// TwinCAT 3 PLC project Controller
// Title: BIO2
// Company: 3P Innovation Ltd.
// Author: James Tyler
// ProgramVersion: 3.1.0.8
// libraries:
//   Standard, * (System)
//   Tc2_ControllerToolbox, * (Beckhoff Automation GmbH)
//   Tc2_Standard, * (Beckhoff Automation GmbH)
//   Tc2_System, * (Beckhoff Automation GmbH)
//   Tc2_TempController, * (Beckhoff Automation GmbH)
//   Tc2_Utilities, * (Beckhoff Automation GmbH)
//   Tc2_XmlDataSrv, * (Beckhoff Automation GmbH)
//   Tc3_Interfaces, * (Beckhoff Automation GmbH)
//   Tc3_Module, * (Beckhoff Automation GmbH)
//   Tc_Persistent, * (Red Rock Controls Limited)
//   Tc2_MC2,newest,Beckhoff Automation GmbH
//   Tc_Collections,1.0.0.8,Red Rock Controls
//   Tc_Helper,1.0.0.8,Red Rock Controls
// project tree:
//   Classes/Compress/ FB_Compress.TcPOU
//   Classes/Config/ TConfig.TcPOU, TConfigData.TcDUT
//   Classes/Pusher/ FB_Pusher.TcPOU
//   Classes/Shield/ FB_Shield.TcPOU
//   DUTs/ E_LampState.TcDUT (not stored), E_CTRL_STATE.TcDUT, Limits.TcDUT, Recipe.TcDUT, Rec_Compress.TcDUT, Rec_Other.TcDUT, Rec_Pusher.TcDUT, Rec_Clamp.TcDUT (not stored), Rec_Shield.TcDUT
//   GVLs/ GVL_IO.TcGVL, GVL_Objects.TcGVL, GVL_ZenOn.TcGVL
//   / PlcTask.TcTTO, Task_Fast.TcTTO
//   POUs/ Config_Slow.TcPOU, FB_AxisControl.TcPOU, FB_LampController.TcPOU, F_DisplayText.TcPOU (not stored), PRG_MAIN.TcPOU, PRG_IO.TcPOU, PRG_Machine.TcPOU
//   XML/ eXMLState.TcDUT, FB_Retain.TcPOU, FB_RetainedData.TcPOU (not stored)
// real-time tasks:
//   TASK PlcTask: cycle T#10ms, priority 20, ADS port 350
//   TASK Task_Fast: cycle T#1ms, priority 21, ADS port 351
// motion (NC):
//   TASK NC-Task 1 SAF: cycle T#2ms, priority 4, ADS port 501
//   TASK NC-Task 1 SVB: cycle T#10ms, priority 8, ADS port 511
//   AXIS Compress (id 1)
//     Dynamic: Acceleration=60.7875, Deceleration=60.7875, Jerk=182.363
//     Velo: RefSearch=0.40525, RefSync=0.40525, SlowManual=2.02625, FastManual=12.1575, Fast=40.525, Maximum=200
//     OtherSettings: AllowMotionCmdToSlave=true
//     encoder EncType=19
//       EncPara: ScaleFactorNumerator=0.5, ScaleFactorDenominator=1048576, ModuloFactor=0.5, MaxCount=#xffffffff
//     drive DrvType=16
//       DrvPara: MaxCount=#xffffffff
//         Analog: VeloReferenz=200, VeloScale=32
//         TimeComp: TaskDelayCycles=1
//     controller CtrType=1
//       CtrPara: PriorControlFactor=1
//         PosDiffControl: Enable=false, Range=0.05
//         PID: PosKp=20
//         Observer: BandWidth=20
//   AXIS Pusher (id 2)
//     Dynamic: Acceleration=60.7875, Deceleration=60.7875, Jerk=182.3625
//     Velo: RefSearch=0.40525, RefSync=0.40525, SlowManual=2.02625, FastManual=12.1575, Fast=40.525, Maximum=40.525
//     OtherSettings: AllowMotionCmdToSlave=true
//     encoder EncType=19
//       EncPara: ScaleFactorNumerator=0.5, ScaleFactorDenominator=1048576, ModuloFactor=0.5, MaxCount=#xffffffff
//     drive DrvType=16
//       DrvPara: MaxCount=#xffffffff
//         Analog: VeloReferenz=100, VeloScale=32
//         TimeComp: TaskDelayCycles=1
//     controller CtrType=1
//       CtrPara: PriorControlFactor=1
//         PosDiffControl: Enable=false, Range=0.5
//         PID: PosKp=20
//         Observer: BandWidth=20
//   AXIS Shield (id 3)
//     Dynamic: Acceleration=60.7875, Deceleration=60.7875, Jerk=182.363
//     Velo: RefSearch=0.40525, RefSync=0.40525, SlowManual=2.02625, FastManual=12.1575, Fast=200, Maximum=200
//     OtherSettings: AllowMotionCmdToSlave=true
//     encoder EncType=19
//       EncPara: ScaleFactorNumerator=0.5, ScaleFactorDenominator=1048576, ModuloFactor=0.5, MaxCount=#xffffffff
//     drive DrvType=16
//       DrvPara: MaxCount=#xffffffff
//         Analog: VeloReferenz=200, VeloScale=32
//         TimeComp: TaskDelayCycles=1
//     controller CtrType=1
//       CtrPara: PriorControlFactor=1
//         PosDiffControl: Enable=false, Range=0.05
//         PID: PosKp=20
//         Observer: BandWidth=20
// I/O:
//   DEVICE Device 1 (EtherCAT), AmsNetId 5.47.207.20.2.1
//     Term 5 (EK1100) [EK1100 EtherCAT Coupler (2A E-Bus)]
//       Term 6 (EL1809) [EL1809 16Ch. Dig. Input 24V, 3ms]
//       Term 7 (EL2798) [EL2798 8Ch. Dig. Output 24V AC/DC, 2A, potential-free]
//       Term 13 (EL9011) [EL9011 End Terminal]
//     Term 8 (EK1100) [EK1100 EtherCAT Coupler (2A E-Bus)]
//       Term 9 (EL7201-9014) [EL7201-9014 1Ch. MDP742 Servo motor output stage with OCT (50V, 4A) and STO input]
//       Term 10 (EL7201-9014) [EL7201-9014 1Ch. MDP742 Servo motor output stage with OCT (50V, 4A)  and STO input]
//       Term 11 (EL7201-9014) [EL7201-9014 1Ch. MDP742 Servo motor output stage with OCT (50V, 4A)  and STO input]
//       Term 12 (EL1809) [EL1809 16Ch. Dig. Input 24V, 3ms]
//       Term 14 (EL9011) [EL9011 End Terminal]
//   DEVICE Device 3 (RT-Ethernet Protocol) (disabled), AmsNetId 5.47.207.20.4.1
// variable links:
//   NC-Task 1 SAF/Axes/Compress <-> Device 1 (EtherCAT)/Term 8 (EK1100)/Term 9 (EL7201-9014)
//     Drive/Inputs/In/nDcOutputTime <-> InfoData/DcOutputShift
//     Drive/Inputs/In/nState1 <-> DRV Statusword/Statusword
//     Drive/Inputs/In/nState2 <-> DRV Statusword/Statusword @bit 8
//     Drive/Inputs/In/nState4 @bit 1 <-> WcState/InputToggle
//     Drive/Inputs/In/nState4 <-> WcState/WcState
//     Drive/Outputs/Out/nCtrl1 <-> DRV Controlword/Controlword
//     Drive/Outputs/Out/nCtrl2 <-> DRV Controlword/Controlword @bit 8
//     Drive/Outputs/Out/nDataOut2 <-> DRV Target velocity/Target velocity
//     Enc/Inputs/In/nDataIn1 <-> FB Position/Position
//     Enc/Inputs/In/nDcInputTime <-> InfoData/DcInputShift
//     Enc/Inputs/In/nState4 @bit 1 <-> WcState/InputToggle
//     Enc/Inputs/In/nState4 <-> WcState/WcState
//   NC-Task 1 SAF/Axes/Pusher <-> Device 1 (EtherCAT)/Term 8 (EK1100)/Term 10 (EL7201-9014)
//     Drive/Inputs/In/nDcOutputTime <-> InfoData/DcOutputShift
//     Drive/Inputs/In/nState1 <-> DRV Statusword/Statusword
//     Drive/Inputs/In/nState2 <-> DRV Statusword/Statusword @bit 8
//     Drive/Inputs/In/nState4 @bit 1 <-> WcState/InputToggle
//     Drive/Inputs/In/nState4 <-> WcState/WcState
//     Drive/Outputs/Out/nCtrl1 <-> DRV Controlword/Controlword
//     Drive/Outputs/Out/nCtrl2 <-> DRV Controlword/Controlword @bit 8
//     Drive/Outputs/Out/nDataOut2 <-> DRV Target velocity/Target velocity
//     Enc/Inputs/In/nDataIn1 <-> FB Position/Position
//     Enc/Inputs/In/nDcInputTime <-> InfoData/DcInputShift
//     Enc/Inputs/In/nState4 @bit 1 <-> WcState/InputToggle
//     Enc/Inputs/In/nState4 <-> WcState/WcState
//   NC-Task 1 SAF/Axes/Shield <-> Device 1 (EtherCAT)/Term 8 (EK1100)/Term 11 (EL7201-9014)
//     Drive/Inputs/In/nDcOutputTime <-> InfoData/DcOutputShift
//     Drive/Inputs/In/nState1 <-> DRV Statusword/Statusword
//     Drive/Inputs/In/nState2 <-> DRV Statusword/Statusword @bit 8
//     Drive/Inputs/In/nState4 @bit 1 <-> WcState/InputToggle
//     Drive/Inputs/In/nState4 <-> WcState/WcState
//     Drive/Outputs/Out/nCtrl1 <-> DRV Controlword/Controlword
//     Drive/Outputs/Out/nCtrl2 <-> DRV Controlword/Controlword @bit 8
//     Drive/Outputs/Out/nDataOut2 <-> DRV Target velocity/Target velocity
//     Enc/Inputs/In/nDataIn1 <-> FB Position/Position
//     Enc/Inputs/In/nDcInputTime <-> InfoData/DcInputShift
//     Enc/Inputs/In/nState4 @bit 1 <-> WcState/InputToggle
//     Enc/Inputs/In/nState4 <-> WcState/WcState
//   Controller/Controller Instance <-> Device 1 (EtherCAT)/Term 5 (EK1100)/Term 6 (EL1809)
//     PlcTask Inputs/GVL_IO.ixCabinetE_StopButtonOkay <-> Channel 1/Cabinet E-Stop
//     PlcTask Inputs/GVL_IO.ixE_StopRelayOkay <-> Channel 2/Input
//     PlcTask Inputs/GVL_IO.ixGuardRelayOkay <-> Channel 3/Input
//     PlcTask Inputs/GVL_IO.ixResetButton <-> Channel 6/Input
//     PlcTask Inputs/GVL_IO.ixStartButton <-> Channel 9/Input
//     PlcTask Inputs/GVL_IO.ixStop_Button <-> Channel 10/Input
//     Task_Fast Inputs/GVL_IO.ixSpareIN4 <-> Channel 4/Input
//     Task_Fast Inputs/GVL_IO.ixSpareIN5 <-> Channel 5/Input
//     Task_Fast Inputs/GVL_IO.ixSpareIN7 <-> Channel 7/Input
//     Task_Fast Inputs/GVL_IO.ixSpareIN8 <-> Channel 8/Input
//   Controller/Controller Instance <-> Device 1 (EtherCAT)/Term 5 (EK1100)/Term 7 (EL2798)
//     PlcTask Outputs/GVL_IO.qxClamp <-> Channel 2/Output
//     PlcTask Outputs/GVL_IO.qxEnableE_Stop <-> Channel 1/Output
//     PlcTask Outputs/GVL_IO.qxResetButtonLamp <-> Channel 5/Output
//     PlcTask Outputs/GVL_IO.qxStartButtonLamp <-> Channel 4/Output
//     Task_Fast Outputs/GVL_IO.qxSpareOUT3 <-> Channel 3/Output
//   Controller/Controller Instance <-> Device 1 (EtherCAT)/Term 8 (EK1100)/Term 12 (EL1809)
//     PlcTask Inputs/GVL_IO.ixCompressHomeSwitch <-> Channel 1/Input
//     PlcTask Inputs/GVL_IO.ixGuardOkay <-> Channel 9/Input
//     PlcTask Inputs/GVL_IO.ixMachineE_StopButtonOkay <-> Channel 10/Input
//     PlcTask Inputs/GVL_IO.ixPusherHomeSwitch <-> Channel 3/Input
//     PlcTask Inputs/GVL_IO.ixShieldHomeSwitch <-> Channel 5/Input
//     PlcTask Inputs/GVL_IO.ixStart_Button_Machine <-> Channel 7/Input
//     Task_Fast Inputs/GVL_IO.ixFanCartridgeDiagnostics <-> Channel 11/Input
//   Controller/Controller Instance <-> NC-Task 1 SAF/Axes/Compress
//     PlcTask Inputs/GVL_IO.CompressAxis.NcToPlc <-> Outputs/ToPlc
//     PlcTask Outputs/GVL_IO.CompressAxis.PlcToNc <-> Inputs/FromPlc
//   Controller/Controller Instance <-> NC-Task 1 SAF/Axes/Pusher
//     PlcTask Inputs/GVL_IO.PusherAxis.NcToPlc <-> Outputs/ToPlc
//     PlcTask Outputs/GVL_IO.PusherAxis.PlcToNc <-> Inputs/FromPlc
//   Controller/Controller Instance <-> NC-Task 1 SAF/Axes/Shield
//     PlcTask Inputs/GVL_IO.ShieldAxis.NcToPlc <-> Outputs/ToPlc
//     PlcTask Outputs/GVL_IO.ShieldAxis.PlcToNc <-> Inputs/FromPlc

CONFIGURATION Controller
    RESOURCE PLC ON TwinCAT3
        TASK PlcTask(INTERVAL := T#10ms, PRIORITY := 20);
        TASK Task_Fast(INTERVAL := T#1ms, PRIORITY := 21);
        PROGRAM PRG_MAIN WITH PlcTask : PRG_MAIN;
        PROGRAM Config_Slow WITH Task_Fast : Config_Slow;
    END_RESOURCE
END_CONFIGURATION

// ---- Classes/Config/TConfigData.TcDUT
{attribute 'pack_mode' := '0'}
TYPE TConfigData :
STRUCT
	
	//Limits
	con_max_limit_Compress 					:LREAL;
	con_max_limit_Shield 					:LREAL;
	con_max_limit_Pusher 					:LREAL;
	con_max_pusher_shield_diff				:LREAL;
	
	//Rec1_Name        						:STRING;
	Rec1_Name_1								:UDINT;
	Rec1_Name_2								:UDINT;
	Rec1_Name_3								:UDINT;
	Rec1_Name_4								:UDINT;
	Rec1_Name_5								:UDINT;
	
	Rec1_Shield_Retract_Speed				:LREAL;
	Rec1_Shield_Initial_Speed				:LREAL;
	Rec1_Shield_Initial_Distance			:LREAL;
	Rec1_Compress_Initial_Speed				:LREAL;
	Rec1_Compress_Initial_Distance			:LREAL;
	Rec1_Compress_Shield_Dwell				:LREAL;
	Rec1_Compress_Relax_Distance			:LREAL;
	Rec1_Compress_Retract_Speed				:LREAL;
	Rec1_Pusher_Initial_Speed				:LREAL;
	Rec1_Pusher_Initial_Distance			:LREAL;
	Rec1_Pusher_Eject_Speed					:LREAL;
	Rec1_Pusher_Eject_Distance				:LREAL;
	Rec1_Pusher_Retract_Speed				:LREAL;
	Rec1_Pusher_tamp_initial_Speed			:LREAL;
	Rec1_Pusher_tamp_initial_distance		:LREAL;
	Rec1_Pusher_tamp_final_Speed			:LREAL;
	Rec1_Pusher_tamp_final_distance			:LREAL;
	Other1_Compress_Home_Offset				:LREAL;
	Other1_Pusher_Home_Offset				:LREAL;
	Other1_Shield_Home_Offset				:LREAL;
	Other1_Axis_Acceleration				:LREAL;
	Other1_Axis_Deceleration				:LREAL;
	Other1_Axis_Jerk						:LREAL;
	Other1_Memory_Free						:LREAL;
	Clamp1_Release_Instance					:LREAL;	
	
	//Rec2_Name        						:STRING;
	Rec2_Name_1								:UDINT;
	Rec2_Name_2								:UDINT;
	Rec2_Name_3								:UDINT;
	Rec2_Name_4								:UDINT;
	Rec2_Name_5								:UDINT;
	
	Rec2_Shield_Retract_Speed				:LREAL;
	Rec2_Shield_Initial_Speed				:LREAL;
	Rec2_Shield_Initial_Distance			:LREAL;
	Rec2_Compress_Initial_Speed				:LREAL;
	Rec2_Compress_Initial_Distance			:LREAL;
	Rec2_Compress_Shield_Dwell				:LREAL;
	Rec2_Compress_Relax_Distance			:LREAL;
	Rec2_Compress_Retract_Speed				:LREAL;
	Rec2_Pusher_Initial_Speed				:LREAL;
	Rec2_Pusher_Initial_Distance			:LREAL;
	Rec2_Pusher_Eject_Speed					:LREAL;
	Rec2_Pusher_Eject_Distance				:LREAL;
	Rec2_Pusher_Retract_Speed				:LREAL;
	Rec2_Pusher_tamp_initial_Speed			:LREAL;
	Rec2_Pusher_tamp_initial_distance		:LREAL;
	Rec2_Pusher_tamp_final_Speed			:LREAL;
	Rec2_Pusher_tamp_final_distance			:LREAL;
	Other2_Compress_Home_Offset				:LREAL;
	Other2_Pusher_Home_Offset				:LREAL;
	Other2_Shield_Home_Offset				:LREAL;
	Other2_Axis_Acceleration				:LREAL;
	Other2_Axis_Deceleration				:LREAL;
	Other2_Axis_Jerk						:LREAL;
	Other2_Memory_Free						:LREAL;
	Clamp2_Release_Instance					:LREAL;
	
	//Rec3_Name        						:STRING;
	Rec3_Name_1								:UDINT;
	Rec3_Name_2								:UDINT;
	Rec3_Name_3								:UDINT;
	Rec3_Name_4								:UDINT;
	Rec3_Name_5								:UDINT;
	
	Rec3_Shield_Retract_Speed				:LREAL;
	Rec3_Shield_Initial_Speed				:LREAL;
	Rec3_Shield_Initial_Distance			:LREAL;
	Rec3_Compress_Initial_Speed				:LREAL;
	Rec3_Compress_Initial_Distance			:LREAL;
	Rec3_Compress_Shield_Dwell				:LREAL;
	Rec3_Compress_Relax_Distance			:LREAL;
	Rec3_Compress_Retract_Speed				:LREAL;
	Rec3_Pusher_Initial_Speed				:LREAL;
	Rec3_Pusher_Initial_Distance			:LREAL;
	Rec3_Pusher_Eject_Speed					:LREAL;
	Rec3_Pusher_Eject_Distance				:LREAL;
	Rec3_Pusher_Retract_Speed				:LREAL;
	Rec3_Pusher_tamp_initial_Speed			:LREAL;
	Rec3_Pusher_tamp_initial_distance		:LREAL;
	Rec3_Pusher_tamp_final_Speed			:LREAL;
	Rec3_Pusher_tamp_final_distance			:LREAL;	
	Other3_Compress_Home_Offset				:LREAL;
	Other3_Pusher_Home_Offset				:LREAL;
	Other3_Shield_Home_Offset				:LREAL;
	Other3_Axis_Acceleration				:LREAL;
	Other3_Axis_Deceleration				:LREAL;
	Other3_Axis_Jerk						:LREAL;
	Other3_Memory_Free						:LREAL;	
	Clamp3_Release_Instance					:LREAL;
	
	//Rec4_Name        						:STRING;
	Rec4_Name_1								:UDINT;
	Rec4_Name_2								:UDINT;
	Rec4_Name_3								:UDINT;
	Rec4_Name_4								:UDINT;
	Rec4_Name_5								:UDINT;
	
	Rec4_Shield_Retract_Speed				:LREAL;
	Rec4_Shield_Initial_Speed				:LREAL;
	Rec4_Shield_Initial_Distance			:LREAL;
	Rec4_Compress_Initial_Speed				:LREAL;
	Rec4_Compress_Initial_Distance			:LREAL;
	Rec4_Compress_Shield_Dwell				:LREAL;
	Rec4_Compress_Relax_Distance			:LREAL;
	Rec4_Compress_Retract_Speed				:LREAL;
	Rec4_Pusher_Initial_Speed				:LREAL;
	Rec4_Pusher_Initial_Distance			:LREAL;
	Rec4_Pusher_Eject_Speed					:LREAL;
	Rec4_Pusher_Eject_Distance				:LREAL;
	Rec4_Pusher_Retract_Speed				:LREAL;
	Rec4_Pusher_tamp_initial_Speed			:LREAL;
	Rec4_Pusher_tamp_initial_distance		:LREAL;
	Rec4_Pusher_tamp_final_Speed			:LREAL;
	Rec4_Pusher_tamp_final_distance			:LREAL;
	Other4_Compress_Home_Offset				:LREAL;
	Other4_Pusher_Home_Offset				:LREAL;
	Other4_Shield_Home_Offset				:LREAL;
	Other4_Axis_Acceleration				:LREAL;
	Other4_Axis_Deceleration				:LREAL;
	Other4_Axis_Jerk						:LREAL;
	Other4_Memory_Free						:LREAL;		
	Clamp4_Release_Instance					:LREAL;
	
	//Rec5_Name        						:STRING;
	Rec5_Name_1								:UDINT;
	Rec5_Name_2								:UDINT;
	Rec5_Name_3								:UDINT;
	Rec5_Name_4								:UDINT;
	Rec5_Name_5								:UDINT;
	
	Rec5_Shield_Retract_Speed				:LREAL;
	Rec5_Shield_Initial_Speed				:LREAL;
	Rec5_Shield_Initial_Distance			:LREAL;
	Rec5_Compress_Initial_Speed				:LREAL;
	Rec5_Compress_Initial_Distance			:LREAL;
	Rec5_Compress_Shield_Dwell				:LREAL;
	Rec5_Compress_Relax_Distance			:LREAL;
	Rec5_Compress_Retract_Speed				:LREAL;
	Rec5_Pusher_Initial_Speed				:LREAL;
	Rec5_Pusher_Initial_Distance			:LREAL;
	Rec5_Pusher_Eject_Speed					:LREAL;
	Rec5_Pusher_Eject_Distance				:LREAL;
	Rec5_Pusher_Retract_Speed				:LREAL;
	Rec5_Pusher_tamp_initial_Speed			:LREAL;
	Rec5_Pusher_tamp_initial_distance		:LREAL;
	Rec5_Pusher_tamp_final_Speed			:LREAL;
	Rec5_Pusher_tamp_final_distance			:LREAL;
	Other5_Compress_Home_Offset				:LREAL;
	Other5_Pusher_Home_Offset				:LREAL;
	Other5_Shield_Home_Offset				:LREAL;
	Other5_Axis_Acceleration				:LREAL;
	Other5_Axis_Deceleration				:LREAL;
	Other5_Axis_Jerk						:LREAL;
	Other5_Memory_Free						:LREAL;		
	Clamp5_Release_Instance					:LREAL;
	
	//Rec6_Name        						:STRING;
	Rec6_Name_1								:UDINT;
	Rec6_Name_2								:UDINT;
	Rec6_Name_3								:UDINT;
	Rec6_Name_4								:UDINT;
	Rec6_Name_5								:UDINT;
	
	Rec6_Shield_Retract_Speed				:LREAL;
	Rec6_Shield_Initial_Speed				:LREAL;
	Rec6_Shield_Initial_Distance			:LREAL;
	Rec6_Compress_Initial_Speed				:LREAL;
	Rec6_Compress_Initial_Distance			:LREAL;
	Rec6_Compress_Shield_Dwell				:LREAL;
	Rec6_Compress_Relax_Distance			:LREAL;
	Rec6_Compress_Retract_Speed				:LREAL;
	Rec6_Pusher_Initial_Speed				:LREAL;
	Rec6_Pusher_Initial_Distance			:LREAL;
	Rec6_Pusher_Eject_Speed					:LREAL;
	Rec6_Pusher_Eject_Distance				:LREAL;
	Rec6_Pusher_Retract_Speed				:LREAL;
	Rec6_Pusher_tamp_initial_Speed			:LREAL;
	Rec6_Pusher_tamp_initial_distance		:LREAL;
	Rec6_Pusher_tamp_final_Speed			:LREAL;
	Rec6_Pusher_tamp_final_distance			:LREAL;
	Other6_Compress_Home_Offset				:LREAL;
	Other6_Pusher_Home_Offset				:LREAL;
	Other6_Shield_Home_Offset				:LREAL;
	Other6_Axis_Acceleration				:LREAL;
	Other6_Axis_Deceleration				:LREAL;
	Other6_Axis_Jerk						:LREAL;
	Other6_Memory_Free						:LREAL;		
	Clamp6_Release_Instance					:LREAL;
	
	//Rec7_Name        						:STRING;
	Rec7_Name_1								:UDINT;
	Rec7_Name_2								:UDINT;
	Rec7_Name_3								:UDINT;
	Rec7_Name_4								:UDINT;
	Rec7_Name_5								:UDINT;
	
	Rec7_Shield_Retract_Speed				:LREAL;
	Rec7_Shield_Initial_Speed				:LREAL;
	Rec7_Shield_Initial_Distance			:LREAL;
	Rec7_Compress_Initial_Speed				:LREAL;
	Rec7_Compress_Initial_Distance			:LREAL;
	Rec7_Compress_Shield_Dwell				:LREAL;
	Rec7_Compress_Relax_Distance			:LREAL;
	Rec7_Compress_Retract_Speed				:LREAL;
	Rec7_Pusher_Initial_Speed				:LREAL;
	Rec7_Pusher_Initial_Distance			:LREAL;
	Rec7_Pusher_Eject_Speed					:LREAL;
	Rec7_Pusher_Eject_Distance				:LREAL;
	Rec7_Pusher_Retract_Speed				:LREAL;
	Rec7_Pusher_tamp_initial_Speed			:LREAL;
	Rec7_Pusher_tamp_initial_distance		:LREAL;
	Rec7_Pusher_tamp_final_Speed			:LREAL;
	Rec7_Pusher_tamp_final_distance			:LREAL;
	Other7_Compress_Home_Offset				:LREAL;
	Other7_Pusher_Home_Offset				:LREAL;
	Other7_Shield_Home_Offset				:LREAL;
	Other7_Axis_Acceleration				:LREAL;
	Other7_Axis_Deceleration				:LREAL;
	Other7_Axis_Jerk						:LREAL;
	Other7_Memory_Free						:LREAL;	
	Clamp7_Release_Instance					:LREAL;
	
	//Rec8_Name        						:STRING;
	Rec8_Name_1								:UDINT;
	Rec8_Name_2								:UDINT;
	Rec8_Name_3								:UDINT;
	Rec8_Name_4								:UDINT;
	Rec8_Name_5								:UDINT;
	
	Rec8_Shield_Retract_Speed				:LREAL;
	Rec8_Shield_Initial_Speed				:LREAL;
	Rec8_Shield_Initial_Distance			:LREAL;
	Rec8_Compress_Initial_Speed				:LREAL;
	Rec8_Compress_Initial_Distance			:LREAL;
	Rec8_Compress_Shield_Dwell				:LREAL;
	Rec8_Compress_Relax_Distance			:LREAL;
	Rec8_Compress_Retract_Speed				:LREAL;
	Rec8_Pusher_Initial_Speed				:LREAL;
	Rec8_Pusher_Initial_Distance			:LREAL;
	Rec8_Pusher_Eject_Speed					:LREAL;
	Rec8_Pusher_Eject_Distance				:LREAL;
	Rec8_Pusher_Retract_Speed				:LREAL;
	Rec8_Pusher_tamp_initial_Speed			:LREAL;
	Rec8_Pusher_tamp_initial_distance		:LREAL;
	Rec8_Pusher_tamp_final_Speed			:LREAL;
	Rec8_Pusher_tamp_final_distance			:LREAL;
	Other8_Compress_Home_Offset				:LREAL;
	Other8_Pusher_Home_Offset				:LREAL;
	Other8_Shield_Home_Offset				:LREAL;
	Other8_Axis_Acceleration				:LREAL;
	Other8_Axis_Deceleration				:LREAL;
	Other8_Axis_Jerk						:LREAL;
	Other8_Memory_Free						:LREAL;	
	Clamp8_Release_Instance					:LREAL;
	
	//Rec9_Name        						:STRING;
	Rec9_Name_1								:UDINT;
	Rec9_Name_2								:UDINT;
	Rec9_Name_3								:UDINT;
	Rec9_Name_4								:UDINT;
	Rec9_Name_5								:UDINT;
	
	Rec9_Shield_Retract_Speed				:LREAL;
	Rec9_Shield_Initial_Speed				:LREAL;
	Rec9_Shield_Initial_Distance			:LREAL;
	Rec9_Compress_Initial_Speed				:LREAL;
	Rec9_Compress_Initial_Distance			:LREAL;
	Rec9_Compress_Shield_Dwell				:LREAL;
	Rec9_Compress_Relax_Distance			:LREAL;
	Rec9_Compress_Retract_Speed				:LREAL;
	Rec9_Pusher_Initial_Speed				:LREAL;
	Rec9_Pusher_Initial_Distance			:LREAL;
	Rec9_Pusher_Eject_Speed					:LREAL;
	Rec9_Pusher_Eject_Distance				:LREAL;
	Rec9_Pusher_Retract_Speed				:LREAL;
	Rec9_Pusher_tamp_initial_Speed			:LREAL;
	Rec9_Pusher_tamp_initial_distance		:LREAL;
	Rec9_Pusher_tamp_final_Speed			:LREAL;
	Rec9_Pusher_tamp_final_distance			:LREAL;
	Other9_Compress_Home_Offset				:LREAL;
	Other9_Pusher_Home_Offset				:LREAL;
	Other9_Shield_Home_Offset				:LREAL;
	Other9_Axis_Acceleration				:LREAL;
	Other9_Axis_Deceleration				:LREAL;
	Other9_Axis_Jerk						:LREAL;
	Other9_Memory_Free						:LREAL;	
	Clamp9_Release_Instance					:LREAL;
	
	//Rec10_Name        					:STRING;
	Rec10_Name_1							:UDINT;
	Rec10_Name_2							:UDINT;
	Rec10_Name_3							:UDINT;
	Rec10_Name_4							:UDINT;
	Rec10_Name_5							:UDINT;
	
	Rec10_Shield_Retract_Speed				:LREAL;
	Rec10_Shield_Initial_Speed				:LREAL;
	Rec10_Shield_Initial_Distance			:LREAL;
	Rec10_Compress_Initial_Speed			:LREAL;
	Rec10_Compress_Initial_Distance			:LREAL;
	Rec10_Compress_Shield_Dwell				:LREAL;
	Rec10_Compress_Relax_Distance			:LREAL;
	Rec10_Compress_Retract_Speed			:LREAL;
	Rec10_Pusher_Initial_Speed				:LREAL;
	Rec10_Pusher_Initial_Distance			:LREAL;
	Rec10_Pusher_Eject_Speed				:LREAL;
	Rec10_Pusher_Eject_Distance				:LREAL;
	Rec10_Pusher_Retract_Speed				:LREAL;
	Rec10_Pusher_tamp_initial_Speed			:LREAL;
	Rec10_Pusher_tamp_initial_distance		:LREAL;
	Rec10_Pusher_tamp_final_Speed			:LREAL;
	Rec10_Pusher_tamp_final_distance		:LREAL;
	Other10_Compress_Home_Offset			:LREAL;
	Other10_Pusher_Home_Offset				:LREAL;
	Other10_Shield_Home_Offset				:LREAL;
	Other10_Axis_Acceleration				:LREAL;
	Other10_Axis_Deceleration				:LREAL;
	Other10_Axis_Jerk						:LREAL;
	Other10_Memory_Free						:LREAL;
	Clamp10_Release_Instance				:LREAL;
	

	
	(*Initialised - MUST BE LAST VARIABLE IN STUCTURE*)
    Initialised : BOOL;
END_STRUCT
END_TYPE

// ---- DUTs/E_CTRL_STATE.TcDUT
TYPE E_CTRL_STATE :
(
   eCTRL_STATE_IDLE      := 0, 
   eCTRL_STATE_PASSIVE := 1, 
   eCTRL_STATE_ACTIVE := 2, 
   eCTRL_STATE_RESET    := 3, 
   eCTRL_STATE_MANUAL := 4, 
   eCTRL_STATE_TUNING := 5, 
   eCTRL_STATE_TUNED    := 6, 
   eCTRL_STATE_SELFTEST := 7, 
   eCTRL_STATE_ERROR    := 8, 
   eCTRL_STATE_SYNC_MOVEMENT := 9 
);
END_TYPE

// ---- DUTs/Limits.TcDUT
TYPE Limits :
	STRUCT
		max_limit_Compress				:LREAL;
		max_limit_Shield				:LREAL;
		max_limit_Pusher 				:LREAL;
		max_pusher_shield_diff			:LREAL;
	END_STRUCT
END_TYPE

// ---- DUTs/Recipe.TcDUT
TYPE Recipe :
	STRUCT
		Name        	:STRING(20);
		Shield      	:Rec_Shield;
		Compress		:Rec_Compress;
		Pusher			:Rec_Pusher;
		Clamp			:Rec_Clamp;
		Other			:Rec_Other;
		Memory_Free		:BOOL := TRUE;
	END_STRUCT
END_TYPE

// ---- DUTs/Rec_Compress.TcDUT
TYPE Rec_Compress :
	STRUCT
		Initial_Speed				:LREAL;
		Initial_Distance			:LREAL;
		Shield_Dwell				:LREAL;
		Relax_Distance				:LREAL;
		Retract_Speed				:LREAL;
	END_STRUCT
END_TYPE

// ---- DUTs/Rec_Other.TcDUT
TYPE Rec_Other :
	STRUCT
		Compress_Home_Offset		:LREAL;
		Pusher_Home_Offset			:LREAL;
		Shield_Home_Offset			:LREAL;
		Axis_Acceleration			:LREAL;
		Axis_Deceleration			:LREAL;
		Axis_Jerk					:LREAL;
	END_STRUCT
END_TYPE

// ---- DUTs/Rec_Pusher.TcDUT
TYPE Rec_Pusher :
	STRUCT
		Initial_Speed				:LREAL;
		Initial_Distance			:LREAL;
		Eject_Speed					:LREAL;
		Eject_Distance				:LREAL;
		Retract_Speed				:LREAL;
		tamp_initial_speed			:LREAL;
		tamp_final_speed			:LREAL;
		tamp_initial_distance		:LREAL;
		tamp_final_distance			:LREAL;
	END_STRUCT
END_TYPE

// ---- DUTs/Rec_Shield.TcDUT
TYPE Rec_Shield :
	STRUCT
		Initial_Speed			:LREAL;
		Initial_Distance		:LREAL;
		Retract_Speed			:LREAL;
	END_STRUCT
END_TYPE

// ---- XML/eXMLState.TcDUT
TYPE eXMLState :
(
	
	eWait,
eResetWrite, 
eWriteData, 
eResetRead, 
eReadData
);
END_TYPE

// ---- GVLs/GVL_IO.TcGVL
VAR_GLOBAL
	CompressAxis :AXIS_REF;	
	PusherAxis :AXIS_REF;	
	ShieldAxis :AXIS_REF;	
	ResetLampController : FB_LampController;
	StartLampController : FB_LampController;
	
	Name_String	AT%IB10 :STRING;
	Name_DINT1	AT%IB10	:DINT;
		
	// Cabinet Digital Inputs 1 - Device 1, Term 2
	ixCabinetE_StopButtonOkay AT%IX0.0 :BOOL;
	ixE_StopRelayOkay AT%IX0.1 :BOOL;
	ixGuardRelayOkay AT%IX0.2 :BOOL;
	ixSpareIN4 AT%IX0.3 :BOOL;
	ixSpareIN5 AT%IX0.4 :BOOL;
	ixResetButton AT%IX0.5 :BOOL;
	ixSpareIN7 AT%IX0.6 :BOOL;
	ixSpareIN8 AT%IX0.7 :BOOL;
	ixStart_Button_Machine AT%IX1.0 :BOOL;
	ixStop_Button AT%IX1.1 :BOOL;
	ixSpareIN11 AT%IX1.2 :BOOL;
	ixSpareIN12 AT%IX1.3 :BOOL;
	ixSpareIN13 AT%IX1.4 :BOOL;
	ixSpareIN14 AT%IX1.5 :BOOL;
	ixSpareIN15 AT%IX1.6 :BOOL;
	ixSpareIN16 AT%IX1.7 :BOOL;
	
	// Cabinet Digital Outputs 1 - Device 1, Term 3
	qxEnableE_Stop AT%QX0.0 :BOOL;
	qxClamp		 AT%QX0.1 :BOOL :=FALSE;
	qxSpareOUT3 AT%QX0.2 :BOOL;
	qxStartButtonLamp AT%QX0.3:BOOL;
	qxResetButtonLamp AT%QX0.4 :BOOL;
	qxSpareOUT6 AT%QX0.5 :BOOL;
	qxSpareOUT7 AT%QX0.6 :BOOL;
	qxSpareOUT8 AT%QX0.7 :BOOL;
	
	// Servo Analogue Inputs 1- Device 2, Term 2
	ibCompressServoTorque AT%IB120 :INT;
	ibCompressServoFollowingError AT%IB124 :DINT;
	qbCompressServoTorqueLimit AT%QB120 :UINT;
	
	// Servo Analogue Inputs 1- Device 2, Term 3
	ibPusherServoTorque AT%IB130 :INT;
	ibPusherServoFollowingError AT%IB134 :DINT;
	qbPusherServoTorqueLimit AT%QB130 :UINT;
	
	// Servo Analogue Inputs 1- Device 2, Term 3
	ibShieldServoTorque AT%IB140 :INT;
	ibShieldServoFollowingError AT%IB144 :DINT;
	qbShieldServoTorqueLimit AT%QB140 :UINT;
	
	// Analogue Inputs - Device 2, Term 4
	(*iiAnalogueIn7_HeaterTemperature AT%IB112 :INT;
	iiAnalogueIn8_UserProbeTemperature AT%IB114 :INT;
	// Status Inputs - Device 2, Term 4
	ixHeaterTC_Error AT%IX2.0 :BOOL;
	ixUserTC_Error AT%IX2.1 :BOOL;*)
	
	// Machine Digital Inputs 1 - Device 2, Term 5
	ixCompressHomeSwitch AT%IX2.0 :BOOL;
	ixPusherHomeSwitch AT%IX2.1 :BOOL;
	ixShieldHomeSwitch AT%IX2.2 :BOOL;
	ixStartButton AT%IX2.3 :BOOL;
	ixSpareIN25 AT%IX2.4 :BOOL;
	ixspareIN26 AT%IX2.5 :BOOL;
	ixspareIN27 AT%IX2.6 :BOOL;
	ixSpareIN28 AT%IX2.7 :BOOL;
	ixGuardOkay AT%IX3.0 :BOOL;
	ixMachineE_StopButtonOkay AT%IX3.1 :BOOL;
	ixFanCartridgeDiagnostics AT%IX3.2 :BOOL;
	ixSpareIN32 AT%IX3.3 :BOOL;
	ixSpareIN33 AT%IX3.4 :BOOL;
	ixSpareIN34 AT%IX3.5 :BOOL;
	ixSpareIN35 AT%IX3.6 :BOOL;
	ixSpareIN36 AT%IX3.7 :BOOL;

	CompressServoErrorID: UDINT;
	PusherServoErrorID: UDINT;	
	ShieldServoErrorID: UDINT;
	
	sSystemStateHi : STRING;
	sSystemStateMed : STRING;
	sSystemStateLo : STRING;
	
END_VAR

// ---- GVLs/GVL_Objects.TcGVL
VAR_GLOBAL
	Clock 						: TClock;
	Config 						: TConfig;
	config_request				:BOOL;
	config_count				:INT;
	List_of_Recipes				: ARRAY[1..10] OF Recipe;
END_VAR

// ---- GVLs/GVL_ZenOn.TcGVL
VAR_GLOBAL
	
	
	overtorque_alarm							:BOOL;

	limits_screen								:Limits;
	limits_save									:Limits;
	save_limits									:BOOL:=FALSE;
	parameter_violation							:BOOL:=FALSE;

	//Mode
	Debug_Mode									:BOOL;
	
	//Recipe on the screen (current one)
	Recipe_Visibility							:ARRAY[1..10] OF BOOL:=[10(FALSE)];  //u are here
	

	
	Recipe_Screen								:Recipe;
	Default_Recipe_Visibility					:BOOL :=FALSE;
		
	//end_of_recipe_on_the_screen
	
	//Maintenance
	Maintenance_Visibility						:BOOL;
	Mode_String									:STRING;
	Stage_Name									:STRING;
	Step_Next									:BOOL;
	Toggle_Clamp								:BOOL;
	Force_Home									:BOOL;
	//end of maintenance
	
	//recipe functions
	SaveRecipe									:BOOL :=FALSE;
	SaveasRecipe								:BOOL :=FALSE;	
	
	
	
	LoadRecipe									:ARRAY[1..10] OF BOOL :=[10(FALSE)];
	Load_Request								:BOOL :=FALSE;
	Save_before_load							:BOOL :=FALSE;
	
	DeleteRecipe								:ARRAY[1..10] OF BOOL :=[10(FALSE)];
	Delete_Request								:BOOL :=FALSE;
	
	

	Saveas_name									:STRING;
	Message										:STRING(300);
	alarm_message								:STRING(300);	
	question									:STRING(300);
	current_recipe_message						:STRING;
	
	//end of recipe functions
	
	sc_CompressServoErrorID: UDINT;
	sc_PusherServoErrorID: UDINT;
	sc_ShieldServoErrorID: UDINT;
	sc_sSystemStateHi: STRING;
	sc_sSystemStateMed: STRING;
	sc_sSystemStateLo: STRING;
	

	
	// Servo Analogue Inputs 1- Device 2, Term 2
	CompressServoTorque          	: INT;
	CompressServoFollowingError		: DINT;
	CompressServoTorqueLimit		: UINT;
	
	// Servo Analogue Inputs 1- Device 2, Term 3
	PusherServoTorque				: INT;
	PusherServoFollowingError		: DINT;
	PusherServoTorqueLimit			: UINT;
	
	// Servo Analogue Inputs 1- Device 2, Term 3
	ShieldServoTorque				: INT;
	ShieldServoFollowingError		: DINT;
	ShieldServoTorqueLimit			: UINT;
		

	
	(* Data For the Main Screen *)
	CurrentProcessState				: STRING;			//Main Screen

	

	
	(* Data For the Settings Screen *)
	CompressDisplay					: LREAL;		//Settings Screen
	PusherDisplay					: LREAL;		//Settings Screen
	ShieldDisplay					: LREAL;
	
	Zenon_Offset_Compress			:BOOL;
	Zenon_Offset_Shield				:BOOL;
	Zenon_Offset_Pusher				:BOOL;
				
	
	(* Digital IO *)
	CabinetE_StopButtonOkay			: BOOL;
	E_StopRelayOkay					: BOOL;
	GuardRelayOkay					: BOOL;
	ResetButton                     : BOOL;
	EnableE_Stop					: BOOL;
	StartButtonLamp					: BOOL;
	ResetButtonLamp					: BOOL;
	
	Clamp_Alarm						:BOOL;
	Clamp_Cooling					:BOOL;
	Clamp_State						:BOOL;
	
	CompressHomeSwitch  			:BOOL;
	PusherHomeSwitch 				:BOOL;
	ShieldHomeSwitch 				:BOOL;
	StartButton 					:BOOL;

	GuardOkay 						:BOOL;
	MachineE_StopButtonOkay 		:BOOL;
	FanCartridgeDiagnostics 		:BOOL;

	ResetLamp						: BOOL;			//Digital IO Screen
	
	LampTest						: BOOL;			//Digital IO Screen

	CompressAxisPosition			: LREAL;		//IO Screen
	PusherAxisPosition				: LREAL;
	ShieldAxisPosition				: LREAL;
	
	(* Top Bar *)
	sSystemState					: STRING;		//Top Bar

END_VAR

// ---- POUs/PRG_MAIN.TcPOU
PROGRAM PRG_MAIN
VAR

	test: BOOL;
	debug: INT;

END_VAR

//Recipes
Clock();


IF Config.Initialised() THEN   
	debug := debug+1;
	PRG_IO();
	PRG_Machine();
END_IF

END_PROGRAM

// ---- POUs/PRG_IO.TcPOU
PROGRAM PRG_IO
VAR
	
	TextTimer: ton;
	Message_timer: ton;
	
	//List_of_Recipes				:ARRAY[1..10] OF Recipe;
	recipe_default				:recipe;
	Current_Recipe				:Recipe;
	//old_recipe					:Recipe;
	empty_recipe				:Recipe;
	current_recipe_no			:INT:=1;
	saveas_recipe_no			:INT;
	load_recipe_no				:INT;
	delete_recipe_no			:INT;
	temp						:INT;
	temp2						:INT;
		
	Initialise					:BOOL := TRUE;
	InitialiseTickCounter		:INT;
	TickCounter					:INT;
	
	save_requested				:BOOL := FALSE;
	
	Pusher_Home					:BOOL;
	Shield_Home					:BOOL;
	Compress_Home				:BOOL;
	
	//violation
	old_recipe					:Recipe;
	old_limits					:Limits;
	zero_violation				:BOOL;
	max_distance_violation		:BOOL;
	max_sh_push_diff_violation	:BOOL;
	
	Message_old					:STRING(300);
	
END_VAR

ResetLampController();
StartLampController();
TextTimer();
Message_timer();

//old_recipe:=current_recipe;

IF Initialise THEN
	InitialiseTickCounter := InitialiseTickCounter + 1;
	IF InitialiseTickCounter = 150 THEN
		Config.CopyConfigRecipiesToGlobal();
	END_IF		
	IF InitialiseTickCounter >= 300 THEN	
	//recipe_screen := List_of_Recipes[1];
		recipe_default.Name:='default 1';
	
		recipe_default.Compress.Initial_Distance:=60;
		recipe_default.Compress.Initial_Speed:=20;
		recipe_default.Compress.Relax_Distance:=5;
		recipe_default.Compress.Retract_Speed:=20;
	
		recipe_default.Pusher.Initial_Distance:=40;
		recipe_default.Pusher.Initial_Speed:=20;
		recipe_default.Pusher.Eject_Distance:=5;
		recipe_default.Pusher.Eject_Speed:=20;
		recipe_default.Pusher.Retract_Speed:=20;
	
		recipe_default.Shield.Retract_Speed:=20;
		recipe_default.Shield.Initial_Distance:=40;
		recipe_default.Shield.Initial_Speed:=20;
		
	
		recipe_default.Memory_Free:=FALSE;
	
		List_of_Recipes[1]:=recipe_default;
		recipe_screen:=List_of_Recipes[1];	
		
		limits_screen:=limits_save;
		
		Message:='Welcome!';
	
		InitialiseTickCounter := 0;
		Initialise := FALSE;
	END_IF		
ELSE
	InitialiseTickCounter := 0;

	current_recipe:=recipe_screen;

	//current_recipe_message:=CONCAT('The current recipe number is ',INT_TO_STRING(Current_recipe_no));
	
	IF current_recipe_no = 1 THEN
		Default_Recipe_Visibility:=FALSE;
	ELSE
		Default_Recipe_Visibility:=TRUE;
	END_IF
	
	FOR	temp := 1 TO 10 DO
		Recipe_Visibility[temp]:=NOT(List_of_Recipes[temp].Memory_Free);
	END_FOR
	
	temp:=1;
END_IF


//violation

IF  recipe_screen.Compress.Initial_Distance =0 OR 
	recipe_screen.Compress.Initial_Speed =0 OR 
	recipe_screen.Compress.Relax_Distance =0 OR 
	recipe_screen.Compress.Retract_Speed =0 OR
	recipe_screen.Pusher.Eject_Distance = 0 OR
	recipe_screen.pusher.Eject_Speed = 0 OR
	recipe_screen.pusher.Initial_Distance = 0 OR
	recipe_screen.Pusher.Initial_Speed = 0 OR
	recipe_screen.Pusher.Retract_Speed = 0 OR
	recipe_screen.Shield.Retract_Speed = 0 THEN
		
	zero_violation := TRUE;
		
	//Message:='Axis Parameters cannot be set to zero';
		
	//recipe_screen := old_recipe;
	//limits_screen := old_limits;
	
ELSE
	zero_violation := FALSE;
END_IF
	
IF 	recipe_screen.Compress.Initial_Distance + recipe_screen.Other.Compress_Home_Offset > limits_screen.max_limit_compress OR
	recipe_screen.Compress.Relax_Distance + recipe_screen.Other.Compress_Home_Offset > limits_screen.max_limit_compress OR
	recipe_screen.Shield.Initial_Distance + recipe_screen.Other.Shield_Home_Offset > limits_screen.max_limit_shield OR
	recipe_screen.Pusher.Initial_Distance + recipe_screen.Other.Pusher_Home_Offset > limits_screen.max_limit_Pusher OR
	recipe_screen.Pusher.tamp_initial_distance + recipe_screen.Other.Pusher_Home_Offset > limits_screen.max_limit_Pusher OR
	recipe_screen.Pusher.tamp_final_distance + recipe_screen.Other.Pusher_Home_Offset > limits_screen.max_limit_Pusher OR
	recipe_screen.Pusher.Eject_Distance + recipe_screen.Other.Pusher_Home_Offset > limits_screen.max_limit_Pusher THEN
		
	max_distance_violation:=TRUE;
		
	//Message:='Maximum Limit Violation';
		
	//recipe_screen := old_recipe;
	//limits_screen := old_limits;
		
ELSE
	max_distance_violation:=FALSE;
END_IF

IF 	(recipe_screen.Other.Pusher_Home_Offset) - (recipe_screen.Other.Shield_Home_Offset) > limits_screen.max_pusher_shield_diff OR
	(recipe_screen.Pusher.Initial_Distance + recipe_screen.Other.Pusher_Home_Offset) - (recipe_screen.Shield.Initial_Distance + recipe_screen.Other.Shield_Home_Offset) > limits_screen.max_pusher_shield_diff OR                      
	(recipe_screen.Pusher.tamp_initial_distance + recipe_screen.Other.Pusher_Home_Offset) - (0 + recipe_screen.Other.Shield_Home_Offset) > limits_screen.max_pusher_shield_diff OR
	(recipe_screen.Pusher.tamp_final_distance + recipe_screen.Other.Pusher_Home_Offset) - (0 + recipe_screen.Other.Shield_Home_Offset) > limits_screen.max_pusher_shield_diff OR
	(recipe_screen.Pusher.Eject_Distance + recipe_screen.Other.Pusher_Home_Offset) - (0 + recipe_screen.Other.Shield_Home_Offset) > limits_screen.max_pusher_shield_diff THEN          
		
	max_sh_push_diff_violation := TRUE;
	
	//Message:='Maximum pusher-shield distance difference violation';
	
	//recipe_screen := old_recipe;
	//limits_screen := old_limits;
		
ELSE
	max_sh_push_diff_violation:=FALSE;
END_IF

IF max_sh_push_diff_violation OR max_distance_violation OR zero_violation THEN
	parameter_violation:=TRUE;
ELSE
	parameter_violation:=FALSE;
END_IF

old_recipe:=recipe_screen;
old_limits:=limits_screen;
//violation end



//alarms
IF zero_violation THEN
	alarm_message:='Some parameters can not be set to zero.'; 
END_IF

IF max_distance_violation THEN
	alarm_message:='Maximum axis distance violation'; 
END_IF

IF max_sh_push_diff_violation THEN
	alarm_message:='Maximum pusher-shield distance difference violation';; 
END_IF

IF Clamp_Alarm THEN
	alarm_message:='Clamp Overtime';
END_IF

IF Overtorque_alarm THEN
	alarm_message:='Motor Overtorque';
END_IF

IF NOT ixGuardOkay THEN
	alarm_message:='Guard Open';
END_IF

IF NOT CabinetE_StopButtonOkay THEN
	alarm_message:='E-Stop Pressed';
END_IF

IF CabinetE_StopButtonOkay AND ixGuardOkay AND NOT parameter_violation AND NOT Overtorque_alarm AND NOT Clamp_Alarm THEN
	alarm_message:='';
END_IF
//end_of_alarms

//save as request
IF SaveasRecipe = TRUE THEN
	saveas_recipe_no:=current_recipe_no;
	WHILE (List_of_Recipes[saveas_recipe_no].Memory_Free = FALSE) AND (saveas_recipe_no<11) DO  
		saveas_recipe_no:=saveas_recipe_no+1;
		
	END_WHILE
	
	IF saveas_recipe_no > 10 THEN
		Message:='Maximum Recipe limit has been reached';
		saveas_recipe_no:=10;
		SaveasRecipe := FALSE;	
	END_IF
		
	IF List_of_Recipes[saveas_recipe_no].Memory_Free = TRUE THEN
		SaveasRecipe:=FALSE;
		
		Message := 'Adding new recipe...';

		List_of_Recipes[saveas_recipe_no]:=current_recipe;
		List_of_Recipes[saveas_recipe_no].Name:=Saveas_name;
		List_of_Recipes[saveas_recipe_no].Memory_Free:=FALSE;
		//current_recipe:=recipe_screen;
		//Config.CopyGlobalRecipiesToConfig();
		
		//Current_Recipe := List_of_Recipes[current_recipe_no];
		//recipe_screen:=current_recipe;

		save_requested := TRUE;		
	
	END_IF
	
END_IF
//save as request end

//load recipe
FOR temp := 1 TO 10 DO
	IF LoadRecipe[temp] = TRUE THEN
		load_recipe_no := temp;
		LoadRecipe[temp] := FALSE;
		
		question := CONCAT('Do you want to save recipe ', recipe_screen.Name);
		question := CONCAT(question,', before loading the recipe ');
		question := CONCAT(question, List_of_Recipes[load_recipe_no].Name);
		question := CONCAT(question,'?'); 
	END_IF
END_FOR

IF Load_Request = TRUE THEN
	
	Load_Request:=FALSE;
	
	IF(Save_before_load=TRUE)THEN
		
		//current_recipe:=recipe_screen;
		List_of_Recipes[current_recipe_no] := current_recipe;
		List_of_Recipes[current_recipe_no].Memory_Free := FALSE;
		//config.CopySettingsFromGlobal();
		Save_before_load := FALSE;
		
		Message := CONCAT('Recipe ',recipe_screen.Name);
		Message := CONCAT(Message,' saving... ');
		
		save_requested := TRUE;	
		
	END_IF
	
	current_recipe_no:=load_recipe_no;
		
	Current_Recipe := List_of_Recipes[current_recipe_no];
	recipe_screen:=current_recipe;
	//Message := CONCAT('Recipe ',current_recipe.Name);
	//Message := CONCAT(Message,' loading... ');

	
END_IF
//load recipe end

//delete recipe
FOR temp := 1 TO 10 DO
	IF DeleteRecipe[temp] = TRUE THEN
		delete_recipe_no := temp;
		DeleteRecipe[temp] := FALSE;
		
		question := CONCAT('Do you want to delete recipe ', List_of_Recipes[delete_recipe_no].Name);
		question := CONCAT(question,'?'); 
	END_IF
END_FOR

IF Delete_Request = TRUE THEN
	
	Delete_Request:=FALSE;
	
	current_recipe_no:=delete_recipe_no;
	
	Message := CONCAT('Recipe ',List_of_Recipes[current_recipe_no].Name );
	Message := CONCAT(Message,' deleting...');
	
	WHILE (delete_recipe_no<10) AND List_of_Recipes[delete_recipe_no+1].Memory_Free = FALSE DO
		List_of_Recipes[delete_recipe_no]:=List_of_Recipes[delete_recipe_no+1];
		delete_recipe_no:=delete_recipe_no+1;
	END_WHILE
	
	List_of_Recipes[delete_recipe_no] := empty_recipe;
	//List_of_Recipes[delete_recipe_no].Memory_Free:=FALSE;
	
	
	IF current_recipe_no = delete_recipe_no AND current_recipe_no <> 1 THEN
		current_recipe_no := current_recipe_no - 1;
	END_IF
		
	Current_Recipe := List_of_Recipes[current_recipe_no];
	recipe_screen:=current_recipe;
	
	save_requested := TRUE;

	
END_IF
//delete recipe end

//save recipe
IF SaveRecipe THEN
	SaveRecipe := FALSE;
	//current_recipe:=recipe_screen;
	//recipe_screen:=current_recipe;
	current_recipe.Memory_Free:=FALSE;
	
	//WHILE (List_of_Recipes[current_recipe_no].Memory_Free = FALSE) AND (current_recipe_no<11) DO  
	//	current_recipe_no:=current_recipe_no+1;
	//END_WHILE
	Message := 'Recipe saving...';	
	
	List_of_Recipes[current_recipe_no] := current_recipe;
	save_requested := TRUE;
	
END_IF
//save recipe end

//save limits
IF save_limits THEN
	save_limits:=FALSE;
	limits_save:=limits_screen;
	save_requested := TRUE;
	Message:='Saving Limits...';
END_IF



IF save_requested = TRUE THEN
	
	save_requested := FALSE;
	Config.CopyGlobalRecipiesToConfig();
	config_request:= TRUE;
	//config_count:=0;
	//Message:='Configuring...';
	
END_IF

//Message Timer
IF Message <> message_old THEN
	Message_timer.IN:=TRUE;
	Message_Timer.PT:=T#10S;
END_IF

IF Message_Timer.Q = TRUE THEN
	Message:='';
	Message_timer.IN:=FALSE;
	//Message_Timer.PT:=T#30S;
END_IF 
Message_old:=Message;
//end of message timer


//Config.CopyGlobalRecipiesToConfig();
//end recipes


(***************************** Data For the Main Screen ***********************)


	(* Settings Page*)


	(* IO Page *)

CabinetE_StopButtonOkay := ixCabinetE_StopButtonOkay;
E_StopRelayOkay:=ixE_StopRelayOkay;
GuardRelayOkay:=ixGuardRelayOkay;
GuardOkay:=ixGuardOkay;

ResetButton := ixResetButton;

		
// Cabinet Digital Outputs 1 - Device 1, Term 3
EnableE_Stop:=qxEnableE_Stop;
	
//StartButtonLamp:=qxStartButtonLamp;
ResetButtonLamp:=qxResetButtonLamp;
	
	
// Servo Analogue Inputs 1- Device 2, Term 2
CompressServoTorque:=ibCompressServoTorque;
CompressServoFollowingError:=ibCompressServoFollowingError;
CompressServoTorqueLimit:=qbCompressServoTorqueLimit;
	
// Servo Analogue Inputs 1- Device 2, Term 3
PusherServoTorque:=ibPusherServoTorque;
PusherServoFollowingError:=ibPusherServoFollowingError;
PusherServoTorqueLimit:=qbPusherServoTorqueLimit;
	
// Servo Analogue Inputs 1- Device 2, Term 3
ShieldServoTorque:=ibShieldServoTorque;
ShieldServoFollowingError:=ibShieldServoFollowingError;
ShieldServoTorqueLimit:=qbShieldServoTorqueLimit;
	

	
// Machine Digital Inputs 1 - Device 2, Term 5
CompressHomeSwitch:=ixCompressHomeSwitch;
PusherHomeSwitch:=ixPusherHomeSwitch;
ShieldHomeSwitch:=ixShieldHomeSwitch;
StartButton:=ixStartButton;
GuardOkay:=ixGuardOkay; 
MachineE_StopButtonOkay:=ixMachineE_StopButtonOkay;
//FanCartridgeDiagnostics:=ixFanCartridgeDiagnostics;

//sc_CompressServoErrorID := CompressServoErrorID;
//sc_PusherServoErrorID := PusherServoErrorID;	
//sc_ShieldServoErrorID := ShieldServoErrorID;
	

//Homed?
Pusher_Home:=PRG_Machine.Pusher.HomeExecuted;
Shield_Home:=PRG_Machine.Shield.HomeExecuted;
Compress_Home:=PRG_Machine.Compress.HomeExecuted;
	
//Clamp
Clamp_State:=qxClamp;

//Mode
IF debug_mode = FALSE THEN
	mode_string:= 'Current Mode: Automatic';
ELSE
	mode_string:= 'Current Mode: Debug';
END_IF

//until here





qxResetButtonLamp := ResetLampController.Q; //io
ResetLamp := ResetLampController.Q; //zenon



ShieldAxisPosition := PRG_Machine.Shield.ShieldServo.fActualPosition;		
PusherAxisPosition := PRG_Machine.Pusher.PusherServo.fActualPosition;
CompressAxisPosition := PRG_Machine.Compress.CompressServo.fActualPosition;

Zenon_Offset_Compress:=PRG_Machine.Compress.OffsetExecuted;
Zenon_Offset_Shield:=PRG_Machine.Shield.OffsetExecuted;
Zenon_Offset_Pusher:=PRG_Machine.Pusher.OffsetExecuted;
		
	(* Top Bar *)
//	sSystemState			: STRING;		//Top Bar
(*		
IF sSystemStateHi = WSTRING_TO_STRING("") THEN
	IF sSystemStateMed = WSTRING_TO_STRING("") THEN
		sSystemState := sSystemStateLo;
	ELSE
		sSystemState := sSystemStateMed;
	END_IF	
ELSE
	sSystemState := sSystemStateHi;
	TextTimer.PT := T#5S;
	TextTimer.IN := TRUE;
	IF TextTimer.Q THEN
		sSystemStateHi :=  WSTRING_TO_STRING("");
		TextTimer.IN := false;
	END_IF
END_IF

sc_sSystemStateHi := sSystemStateHi;
sc_sSystemStateMed := sSystemStateMed;
sc_sSystemStateLo := sSystemStateLo;

*)

PROPERTY List_of_Recipes_config :ARRAY[1..10] OF Recipe;
GET
List_of_Recipes_config := List_of_Recipes;
END_GET
SET
List_of_Recipes := List_of_Recipes_config;
END_SET
END_PROPERTY

PROPERTY recipe_default_ext :Recipe;
GET
recipe_default_ext := recipe_default;
END_GET
SET
recipe_default := recipe_default_ext;
END_SET
END_PROPERTY

END_PROGRAM

// ---- POUs/PRG_Machine.TcPOU
PROGRAM PRG_Machine
VAR
	

	
	//Forced Home
	Forced_Home_State						:INT:=0;
	Forced_Home_State_Next					:INT:=0;
	Forced_Home_Executed					:BOOL:=FALSE;

	//RepetitionCounter: INT;
	
	Pusher :FB_Pusher;
	Compress: FB_Compress;
	Shield: FB_Shield;

	ZenonStart: NT_StartProcess;
	//nameString: STRING;
	
	debug: INT;
	tickcounter: INT;
	tickcounter2: INT;

	State: INT:= 0;
	state_old: INT:=0;
	StateNext: INT:= 0;
	
	SM_StepRequest: BOOL:=FALSE;
	singleStep: BOOL:=FALSE;
		
	Clamp_Security_Time: TIME := T#30S;
	ClampTimer: TON;
	//DwellTimer: TON;
	//SaveTickCounter: INT := 0;

	DatumTaught: BOOL;
	//test: BOOL;
	//ReTeachOffsets: BOOL;
	//StopRequest: BOOL;
	//random: STRING(INT#4);
	rec_temp1: recipe;
	rec_temp2: recipe;
	rec_temp3: recipe;
	
END_VAR

IF TRUE THEN
	debug := debug+1;
END_IF



qbCompressServoTorqueLimit := 1000;
qbPusherServoTorqueLimit := 1000;
qbShieldServoTorqueLimit := 1000;


//The state-machine
CASE State OF
	
0: //Copy config .txt file into machine settings
	


	//Zenon start process function call - appears to never generate errors
	
	//IF ZenonStart.Busy=FALSE THEN
	ZenonStart (
		NETID :=,
		//PATHSTR := 'Hard Disk\CP6606_Runtime\zenonRCE.exe', //'C:\PROGRAM Files\COPA-DATA\zenon 7.20 SP0\Zenrt32.exe',
		//DIRNAME := 'Hard Disk\CP6606_Runtime',  //'C:\Program Files\COPA-DATA\zenon 7.20 SP0',
		PATHSTR := 'Hard Disk\ZenonRunTime\zenonRCE.exe', //'C:\PROGRAM Files\COPA-DATA\zenon 7.20 SP0\Zenrt32.exe',
		DIRNAME := 'Hard Disk\ZenonRunTime',  //'C:\Program Files\COPA-DATA\zenon 7.20 SP0',
		COMNDLINE := '',
		START := TRUE,
		TMOUT := DEFAULT_ADS_TIMEOUT
		);
	StateNext := 10;
	//END_IF	
	
	//IF ZenonStart.BUSY = FALSE THEN
	//	ZenonStart ( START := FALSE );
	//	StateNext := 10;
	//END_IF

10: //When restarting state machine, ensure E-Stop relay is not set
	//PRG_System.fbRecipeHandler.M_Next();
	qxEnableE_Stop := FALSE;
	tickcounter := 0;
	StateNext := 15;
	//qxEnableE_Stop:=TRUE;
15: //Check E-Stop relay is not set then Enable and initialise stuff - disable drive to clear errors
	//u are here
	
	//Shield._Reset();
	//Compress._Reset();
	//Pusher._Reset();
	

	//StartLoad := FALSE;
	ResetLampController.State := off;
	//RepetitionCounter := 0;
	//qxEnableE_Stop := TRUE;
	IF ixCabinetE_StopButtonOkay (*AND ixGuardRelayOkay*) THEN
		qxEnableE_Stop := TRUE;
		StateNext := 20;
	END_IF	
	
20: // Look for E-Stop button reset
	IF ixCabinetE_StopButtonOkay THEN
		ResetLampController.State := steady;
		sSystemStateMed := F_DisplayText("Press RESET button",0);	
		StateNext := 30;
	ELSE
		IF ixCabinetE_StopButtonOkay AND ixMachineE_StopButtonOkay THEN 
			ResetLampController.State := FastFlash;
			sSystemStateMed := F_DisplayText("Guard Open",0);
		ELSE
			ResetLampController.State := off;
			sSystemStateMed := F_DisplayText("E-Stop Depressed",0);
		END_IF
		CurrentProcessState	:= F_DisplayText("not ready",0);	//Main Screen	
	END_IF

30: // Wait for operator to hit reset button
	
	IF ixE_StopRelayOkay THEN
		ResetLampController.State := off;
		StateNext := 40;
		tickcounter := 0;
	ELSE
		tickcounter := tickcounter + 1;
		IF tickcounter >= 9800 THEN
			ResetLampController.State := steady;
			tickcounter := 0;
		END_IF
	END_IF

40: // look for guard closed - disable drive to clear errors
	sSystemStateMed := F_DisplayText("Guard Open",0);	
	CurrentProcessState	:= F_DisplayText("not ready",0);	//Main Screen	

	
	IF NOT ixGuardRelayOkay THEN
		ResetLampController.State := FastFlash;		
	ELSE
		ResetLampController.State := off;
		sSystemStateMed := F_DisplayText("Initialising Axes",0);	
		tickcounter := 0;
		StateNext := 100;
	END_IF
	
100: // wait 2 scans for power supply to drive to stabilise
	tickcounter := tickcounter + 1;
	IF tickcounter >= 2 THEN
		tickcounter := 0;
		StateNext := 110;
	END_IF

110: // prepare for Servo motion - enable drive
//you are here!!!!!!!!!!!!!!!!!!!!!!!!!!!!
	IF NOT ixResetButton THEN
		
		
	
		Shield._Enable();
		Pusher._Enable();
		Compress._Enable();
		
		tickcounter := tickcounter + 1;
		IF tickcounter >= 100 THEN
			tickcounter := 0;

			StateNext := 115;
		END_IF	
	END_IF


	
115: 
	
	//IF Shield.HomeExecuted = FALSE OR Pusher.HomeExecuted = FALSE OR Compress.HomeExecuted = FALSE THEN
	Stage_Name := 'Beginning';
	Maintenance_Visibility:=TRUE;
	qxStartButtonLamp:=TRUE;
	IF (ixStartButton OR Step_Next OR ixStart_Button_Machine) THEN
		IF (parameter_violation = FALSE) THEN
			qxStartButtonLamp:=FALSE;
			StateNext := 119;
			Step_Next := FALSE;
			Clamp_Alarm:=FALSE;
			Maintenance_Visibility:=FALSE;
			Stage_Name := 'Homing and Offsetting';

			rec_temp1:=Shield.Shield_Param;     
			rec_temp2:=Pusher.Pusher_Param;
			rec_temp3:=Compress.Compress_Param; 
		ELSE
			Step_Next:=FALSE;
		END_IF
	END_IF

	
119:
	IF rec_temp1.other.Shield_Home_Offset <> recipe_screen.Other.Shield_Home_Offset THEN
		Shield.HomeExecuted:=FALSE;
		Shield.OffsetExecuted:=FALSE;
	END_IF
	
	IF rec_temp2.other.Pusher_Home_Offset <> recipe_screen.Other.Pusher_Home_Offset THEN
		Pusher.HomeExecuted:=FALSE;
		Pusher.OffsetExecuted:=FALSE;
	END_IF
	
	IF rec_temp3.other.Compress_Home_Offset <> recipe_screen.Other.Compress_Home_Offset THEN
		Compress.HomeExecuted:=FALSE;
		Compress.OffsetExecuted:=FALSE;
	END_IF
	
	Shield.Shield_param:=recipe_screen;
	Compress.Compress_Param := recipe_screen;
	Pusher.Pusher_Param := recipe_screen;
	
	

	IF	Compress.HomeExecuted=FALSE OR Shield.HomeExecuted = FALSE OR Pusher.HomeExecuted = FALSE THEN
		statenext:=120;
	ELSE
		StateNext:=129;
	END_IF
		
120: //you are here!!!!!!!!!!!!

	
	
	IF Pusher.HomeExecuted = FALSE THEN 
		Pusher._Home();
	END_IF
	
	IF Compress.HomeExecuted = FALSE THEN
		Compress._Home();
	END_IF
	
	
	IF Compress.HomeExecuted AND Pusher.HomeExecuted THEN
		StateNext := 125;                //directly to end
		//Compress.HomeExecuted:=FALSE;
		//Pusher.HomeExecuted:=FALSE;
		
	END_IF
	
125:
	//random:='arda';
	IF Shield.HomeExecuted = FALSE THEN
		Shield._Home();
		
	ELSE
		StateNext := 128;
		//Shield.HomeExecuted := FALSE;
	END_IF
128:
		

	IF Compress.OffsetExecuted = FALSE THEN
		Compress.Offset();
	END_IF
	
	IF Shield.OffsetExecuted = FALSE THEN
		Shield.Offset();
	END_IF
	
	IF Pusher.OffsetExecuted = FALSE THEN
		Pusher.Offset();
	END_IF
	
	IF Pusher.OffsetExecuted AND Shield.OffsetExecuted AND Compress.OffsetExecuted THEN
		Maintenance_Visibility := TRUE;
		qxStartButtonLamp:=TRUE;
		IF (ixStartButton OR Step_Next OR ixStart_Button_Machine) THEN
			IF (parameter_violation =FALSE) THEN
				qxStartButtonLamp:=FALSE;
				Shield.Shield_param:=recipe_screen;
				Compress.Compress_Param := recipe_screen;
				Pusher.Pusher_Param := recipe_screen;
			
				StateNext:=130;
				Step_Next:=FALSE;
				Maintenance_Visibility := FALSE;
			ELSE
				Step_Next:=FALSE;
			END_IF
		END_IF
	END_IF
	
	

129: //debug	
	
	IF Debug_Mode THEN
		Maintenance_Visibility := TRUE;
		IF Step_Next THEN
			IF Parameter_Violation = FALSE THEN
				Step_Next:=FALSE;
				StateNext:=130;
				Maintenance_Visibility := FALSE;
			
				Shield.Shield_param:=recipe_screen;
				Compress.Compress_Param := recipe_screen;
				Pusher.Pusher_Param := recipe_screen;
			ELSE
				Step_Next:=FALSE;
			END_IF
		END_IF
	ELSE
		StateNext:=130;
		Maintenance_Visibility := FALSE;
	END_IF
		
130: //stage 1
	Stage_Name := 'Compress Tobacco';
	IF qxClamp = FALSE THEN
		qxClamp:=TRUE;
		ClampTimer.IN:=TRUE;
		ClampTimer.PT:=Clamp_Security_Time;

	END_IF
	
	IF Compress.Stage1Executed = FALSE THEN
		IF state_old = 130 THEN
			Message:='I am trying to continue';
		END_IF 
		Compress._Stage1();
		Compress.HomeExecuted:=FALSE;	
	ELSE
		//Compress.Stage1Executed := FALSE;
		StateNext := 131;
		DatumTaught := FALSE;
	END_IF

131: //debug

	IF Debug_Mode THEN
		Maintenance_Visibility := TRUE;
		IF Step_Next THEN
			IF Parameter_Violation = FALSE THEN
				Step_Next:=FALSE;
				StateNext:=135;
				Maintenance_Visibility := FALSE;
			
				Shield.Shield_param:=recipe_screen;
				Compress.Compress_Param := recipe_screen;
				Pusher.Pusher_Param := recipe_screen;
			ELSE
				Step_Next:=FALSE;
			END_IF
		END_IF
	ELSE
		StateNext:=135;
		Maintenance_Visibility := FALSE;
	END_IF
	
135://stage2
	Stage_Name := 'Load Tobacco';
	Compress.Stage1Executed := FALSE;
	
	IF Pusher.Stage2Executed = FALSE THEN
		Pusher._Stage2();
		Pusher.HomeExecuted:=FALSE;
	END_IF
	
	IF Shield.Stage2Executed = FALSE THEN
		Shield._Stage2();
		Shield.HomeExecuted:=FALSE;
	END_IF
	
	IF Shield.Stage2Executed AND Pusher.Stage2Executed THEN
		//Shield.Stage2Executed:=FALSE;
		//Pusher.Stage2Executed:=FALSE;
		//DatumTaught:=FALSE;
		StateNext := 137;
	END_IF
137: //debug

	IF Debug_Mode THEN
		Maintenance_Visibility := TRUE;
		IF Step_Next THEN
			IF Parameter_Violation = FALSE THEN
				Step_Next:=FALSE;
				StateNext:=140;
				Maintenance_Visibility := FALSE;
			
				Shield.Shield_param:=recipe_screen;
				Compress.Compress_Param := recipe_screen;
				Pusher.Pusher_Param := recipe_screen;
			ELSE
				Step_Next:=FALSE;
			END_IF
		END_IF
	ELSE
		StateNext:=140;
		Maintenance_Visibility := FALSE;
	END_IF
	
140: //stage3
	
	Stage_Name := 'Shield Retract';
	
	Shield.Stage2Executed:=FALSE;
	Pusher.Stage2Executed:=FALSE;
	
	IF	Shield.Stage3Executed = FALSE THEN
		Shield._Stage3();
		Shield.HomeExecuted:=FALSE;	
	ELSE
		//Shield.Stage3Executed := FALSE;
		StateNext := 141;
		DatumTaught := FALSE;
	END_IF

141: //debug

	IF Debug_Mode THEN
		Maintenance_Visibility := TRUE;
		IF Step_Next THEN
			IF Parameter_Violation = FALSE THEN
				Step_Next:=FALSE;
				StateNext:=142;
				Maintenance_Visibility := FALSE;
			
				Shield.Shield_param:=recipe_screen;
				Compress.Compress_Param := recipe_screen;
				Pusher.Pusher_Param := recipe_screen;
			ELSE
				Step_Next:=FALSE;
			END_IF
		END_IF
	ELSE
		StateNext:=142;
		Maintenance_Visibility := FALSE;
	END_IF	
	
142: //Tamp
	
	Stage_Name := 'Tamp';
	
	Shield.Stage3Executed := FALSE;
	
	IF	Pusher.TampExecuted = FALSE THEN
		Pusher.Tamp();
		Pusher.HomeExecuted:=FALSE;	
	ELSE
		StateNext := 143;
	END_IF
	
143: //debug

	IF Debug_Mode THEN
		Maintenance_Visibility := TRUE;
		IF Step_Next THEN
			IF Parameter_Violation = FALSE THEN
				Step_Next:=FALSE;
				StateNext:=145;
				Maintenance_Visibility := FALSE;
			
				Shield.Shield_param:=recipe_screen;
				Compress.Compress_Param := recipe_screen;
				Pusher.Pusher_Param := recipe_screen;
			ELSE
				Step_Next:=FALSE;
			END_IF
		END_IF
	ELSE
		StateNext:=145;
		Maintenance_Visibility := FALSE;
	END_IF
	
145: //stage4
	
	Stage_Name := 'Eject Spill';
	
	Pusher.TampExecuted := FALSE;
	IF	Pusher.Stage4Executed = FALSE THEN
		Pusher._Stage4();
		Pusher.HomeExecuted:=FALSE;	
	ELSE
		//Pusher.Stage4Executed := FALSE;
		StateNext := 147;
		DatumTaught := FALSE;
	END_IF

147: //debug

	IF Debug_Mode THEN
		Maintenance_Visibility := TRUE;
		IF Step_Next THEN
			IF Parameter_Violation = FALSE THEN
				Step_Next:=FALSE;
				StateNext:=150;
				Maintenance_Visibility := FALSE;
			
				Shield.Shield_param:=recipe_screen;
				Compress.Compress_Param := recipe_screen;
				Pusher.Pusher_Param := recipe_screen;
			ELSE
				Step_Next:=FALSE;
			END_IF
		END_IF
	ELSE
		StateNext:=150;
		Maintenance_Visibility := FALSE;
	END_IF
	
150: //stage 5
	
	Stage_Name := 'Retract All';
	
	Pusher.Stage4Executed := FALSE;
	IF Pusher.Stage5Executed = FALSE THEN
		Pusher._Stage5();
		Pusher.HomeExecuted:=FALSE;
	END_IF
	
	IF Compress.Stage5Executed = FALSE THEN
		Compress._Stage5();
		Compress.HomeExecuted:=FALSE;
	END_IF
	
	IF Compress.Stage5Executed AND Pusher.Stage5Executed THEN
		//Compress.Stage5Executed:=FALSE;
		//Pusher.Stage5Executed:=FALSE;
		DatumTaught:=FALSE;
		StateNext := 155;
	END_IF	
151:
	Pusher._Halt();
	Shield._Halt();
	Compress._Halt();
	IF Pusher.PusherServo.xhalted AND Shield.ShieldServo.xHalted AND Compress.CompressServo.xHalted AND (ixStartbutton OR ixStart_Button_Machine) THEN
		Pusher._Halt_false();
		Shield._Halt_false();
		Compress._Halt_false();
		Pusher._Soft_Reset();
		Shield._Soft_Reset();
		Compress._Soft_Reset();
		statenext:=state_old;
	END_IF

155: //end
	Compress.Stage5Executed:=FALSE;
	Pusher.Stage5Executed:=FALSE;
	
	Pusher.HomeExecuted:= TRUE;
	Shield.HomeExecuted:=TRUE;
	Compress.HomeExecuted:=TRUE;
	statenext:= 115;

	
1000: // overtorque
	CurrentProcessState	:= F_DisplayText("Process incomplete",0);			//Main Screen
	//StartLoad := FALSE;
	
	Compress._Reset();
	Pusher._Reset();
	Shield._Reset();
	
	qxclamp:=FALSE;
	ClampTimer.IN:=FALSE;
	ClampTimer.PT:=Clamp_Security_Time;
	
	statenext:=2000;
	
	
	

	
2000: // guard and estop
	
	tickcounter:= tickcounter+1;
	IF	tickcounter = 100 THEN
		tickcounter:=0;
		statenext:=15;
		overtorque_alarm:=FALSE;
	END_IF

2010: // clamp alarm
	
	tickcounter:= tickcounter+1;

	
	IF clamp_alarm THEN
		
		IF	tickcounter = 3000 THEN
			tickcounter:=0;
			statenext:=100;
			Clamp_Cooling := FALSE;
			Clamp_Alarm := FALSE;
		ELSE
			Clamp_Cooling := TRUE;
			
			IF Pusher.PusherServo.xstopped AND Shield.ShieldServo.xstopped AND Compress.CompressServo.xstopped THEN
				Pusher._Reset();
				Shield._Reset();
				Compress._Reset();
			END_IF
		END_IF
	ELSE
		IF	tickcounter = 100 THEN
			tickcounter:=0;
			statenext:=100;
			Clamp_Cooling := FALSE;
		ELSIF Pusher.PusherServo.xstopped AND Shield.ShieldServo.xstopped AND Compress.CompressServo.xstopped THEN
			Pusher._Reset();
			Shield._Reset();
			Compress._Reset();
			
		END_IF
	END_IF
	
2020: //force home
(*	
	IF Forced_Home_Executed = FALSE THEN
		Handle_Forced_Home();	
	ELSE
		StateNext:=115;
		Forced_Home_Executed:=FALSE;
	END_IF
*)
	
END_CASE

Pusher._Update();
Shield._Update();
Compress._Update();
ClampTimer();

IF 	StateNext <> 115 AND 
	StateNext <> 128 THEN
	qxStartButtonLamp:=FALSE;
END_IF

IF 	StateNext <> 115 AND 
	StateNext <> 128 AND 
	StateNext <> 129 AND 
	StateNext <> 131 AND 
	StateNext <> 137 AND 
	StateNext <> 141 AND 
	StateNext <> 143 AND 
	StateNext <> 147 THEN

	Maintenance_Visibility := FALSE;
END_IF

//Motor Overtorque
IF StateNext >= 110 AND StateNext <= 155  THEN					// machine is running
	
	IF ibCompressServoTorque  > 2000 OR ibCompressServoTorque  < -2000 THEN						// PuckSlideServo torque too high
		//Message := WSTRING_TO_STRING("Tobacco Compress Servo over-torque");
		StateNext := 1000;
		tickcounter:=0;
		overtorque_alarm:= TRUE;	
	END_IF
	
	IF ibPusherServoTorque  > 2000 OR ibPusherServoTorque  < -2000 THEN						// HeaterSlideServo torque too high
		//Message := WSTRING_TO_STRING("Rod Pusher Servo over-torque");
		StateNext := 1000;
		tickcounter:=0;
		overtorque_alarm:= TRUE;	
	END_IF
	
	IF ibShieldServoTorque  > 2000 OR ibShieldServoTorque  < -2000 THEN						// HeaterSlideServo torque too high
		//Message := WSTRING_TO_STRING("Rod Shield Servo over-torque");
		StateNext := 1000;
		tickcounter:=0;
		overtorque_alarm:= TRUE;	
	END_IF
END_IF


//Toggole Clamp
IF (StateNext >= 115 AND StateNext <= 155) AND Toggle_Clamp THEN
	Toggle_Clamp := FALSE;
	IF qxClamp = FALSE THEN
		
		qxClamp:=TRUE;
		ClampTimer.IN:=TRUE;
		ClampTimer.PT:=Clamp_Security_Time;

	ELSE
		
		qxClamp:=FALSE;
		ClampTimer.IN:=FALSE;
		ClampTimer.PT:=Clamp_Security_Time;
		
	END_IF
	
	
END_IF

//stop button
IF NOT ixstop_button AND (Statenext<>151) THEN
	//	state_old:=statenext;
	//	statenext:= 151;
	tickcounter:=0;
	//Message:='Clamp Overtime';
	qxClamp:=FALSE;

	
	ClampTimer.IN:=FALSE;
	ClampTimer.PT:=Clamp_Security_Time;
	
	
	
	Compress._mc_stop();
	Shield._mc_stop();
	Pusher._mc_stop();
	StateNext := 2010;
	
	
END_IF

//Clamp Err
IF (Clamptimer.Q=TRUE) AND StateNext >= 100 AND StateNext <= 155 THEN 
	
	tickcounter:=0;
	//Message:='Clamp Overtime';
	qxClamp:=FALSE;

	
	ClampTimer.IN:=FALSE;
	ClampTimer.PT:=Clamp_Security_Time;
	
	Clamp_Alarm:=TRUE;
	
	Compress._mc_stop();
	Shield._mc_stop();
	Pusher._mc_stop();
	StateNext := 2010;

END_IF

//Home
IF (Force_Home) AND StateNext >= 115 AND StateNext <= 155 THEN 
	Force_Home:=FALSE;
	StateNext := 2020;
	tickcounter:=0;
	
	
	
	qxclamp:=FALSE;
	ClampTimer.IN:=FALSE;
	ClampTimer.PT:=Clamp_Security_Time;
	
	Pusher._Reset();
	Shield._Reset();
	Compress._Reset();
END_IF

//guard
IF (NOT ixGuardRelayOkay) AND StateNext >= 100 AND StateNext <= 155 THEN 
	
	StateNext := 2000;
	tickcounter:=0;
	
	//Message:='Guard Open';
	
	qxclamp:=FALSE;
	ClampTimer.IN:=FALSE;
	ClampTimer.PT:=Clamp_Security_Time;
	
	IF Pusher.HomeExecuted= FALSE OR Shield.HomeExecuted = FALSE OR Compress.HomeExecuted = FALSE THEN
		Pusher._Reset();
		Shield._Reset();
		Compress._Reset();
	ELSE
		Pusher._Reset_Medium();
		Shield._Reset_Medium();
		Compress._Reset_Medium();
	END_IF
END_IF

//estop
IF (NOT ixCabinetE_StopButtonOkay) AND StateNext >= 30 AND StateNext <= 155 THEN 
	
	tickcounter:=0;
	
	//Message:='E-stop Pressed';
	
	qxclamp:=FALSE;
	ClampTimer.IN:=FALSE;
	ClampTimer.PT:=Clamp_Security_Time;
	

	
	//IF Compress.CompressServo.xStopped AND Shield.ShieldServo.xStopped AND Pusher.PusherServo.xStopped THEN
	StateNext := 2000;
	Pusher._Reset();
	Shield._Reset();
	Compress._Reset();
	//END_IF
END_IF

//IF State <> StateNext THEN - step through the state machine if required
IF singleStep AND statenext > 119 THEN
	//IF NOT SM_StepRequest THEN
	//	SM_StepRequest := TRUE; 
	//END_IF
	IF SM_StepRequest THEN
		SM_StepRequest := FALSE;
		State := StateNext;
	END_IF
ELSE
	State := StateNext;
END_IF

PROPERTY ext_Clamp_Security_Time : TIME
GET
ext_Clamp_Security_Time := Clamp_Security_Time;
END_GET
SET
Clamp_Security_Time := ext_Clamp_Security_Time;
END_SET
END_PROPERTY

PROPERTY ext_ClampTimer : TON
GET
ext_ClampTimer:=ClampTimer;
END_GET
SET
ClampTimer:=ext_ClampTimer;
END_SET
END_PROPERTY

METHOD Handle_Forced_Home
VAR_INPUT
END_VAR
CASE Forced_Home_State OF
	
0:	
	tickcounter:=tickcounter + 1;
	IF tickcounter = 100 THEN
		Forced_Home_State_Next:=5;
	END_IF
5:	



END_CASE

Forced_Home_State_Next := Forced_Home_State;
END_METHOD

METHOD StopClampTimer
VAR_INPUT
END_VAR
ClampTimer.IN:=FALSE;
ClampTimer.PT:= Clamp_Security_Time;
END_METHOD

END_PROGRAM

// ---- Classes/Pusher/FB_Pusher.TcPOU
FUNCTION_BLOCK FB_Pusher
VAR_INPUT
END_VAR
VAR_OUTPUT
END_VAR
VAR

PusherServo        			:FB_AxisControl;

_Pusher_param				:recipe;



ToolPositioningSpeed	: LREAL := 20;
ToolPositioningAccel	: LREAL := 100;
ToolPositioningJerk		: LREAL := 1000;
ToolHomingSpeed			: LREAL := 2;

PusherServoEnable			:BOOL;
PusherServoEnabled			:BOOL;

_ExecutedHome				:BOOL:=FALSE;
_ExecutedStage2				:BOOL:=FALSE;
_ExecutedStage4				:BOOL:=FALSE;
_ExecutedStage5				:BOOL:=FALSE;
_ExecutedOffset				:BOOL:=FALSE;
_ExecutedTamp				:BOOL:=FALSE;

tickcounter_pusher: 		INT :=0;
State: 						INT:= 0;
StateNext: 					INT:= 0;

pusher_old_position			:LREAL;


END_VAR

METHOD _Enable 
VAR_INPUT
END_VAR

PusherServoEnable := TRUE;
END_METHOD

METHOD _Halt : BOOL
VAR_INPUT
END_VAR
PusherServo.xHalt:=TRUE;
END_METHOD

METHOD _Halt_false : BOOL
VAR_INPUT
END_VAR
PusherServo.xHalt:=FALSE;
END_METHOD

METHOD _Home 
VAR_INPUT
	
END_VAR


VAR


END_VAR

VAR_OUTPUT
	
END_VAR


CASE State OF //you are here



0:	
	_ExecutedHome := FALSE;
	PusherServo.fVelocity := ToolPositioningSpeed;
	PusherServo.fAxisAcceleration := ToolPositioningAccel;
	PusherServo.fAxisDeceleration := ToolPositioningAccel;
	PusherServo.fAxisJerk := ToolPositioningJerk;

	IF ixPusherHomeSwitch THEN
		PusherServo.xPositiveDirection := FALSE;
		IF  tickcounter_pusher < 10 THEN
			tickcounter_pusher := tickcounter_pusher + 1;  // can be put in onditional
		
		ELSE
		//IF tickcounter_compress >= 10 THEN
			PusherServo.xMoveV := TRUE;
		END_IF
	ELSE
	
		//CompressServo.xHalt := NOT CompressServo.xHalt;
		PusherServo.xMoveV := FALSE;
		//CompressServo.xHalt := NOT CompressServo.xHalt;
		PusherServo.xHalt := TRUE;
		IF PusherServo.xHalted THEN
			tickcounter_pusher:=0;
			StateNext := 5;
		END_IF
	
	END_IF
	
5:
	
	PusherServo.xHalt := FALSE;
	tickcounter_Pusher := tickcounter_Pusher + 1;
	IF tickcounter_Pusher >= 10 THEN
		tickcounter_Pusher := 0;
		StateNext := 10;
	END_IF
	
10:
	PusherServo.fVelocity := ToolHomingSpeed;
	
	IF NOT ixPusherHomeSwitch THEN
		PusherServo.xPositiveDirection := TRUE;
		IF tickcounter_Pusher < 10 THEN
			tickcounter_Pusher := tickcounter_Pusher + 1;
		ELSE
		//IF tickcounter >= 10 THEN
			PusherServo.xMoveV := TRUE;
		END_IF
	ELSE
		PusherServo.xMoveV := FALSE;
		PusherServo.xHalt := TRUE;
		IF PusherServo.xHalted THEN
			tickcounter_Pusher := 0;
			StateNext := 15;
		END_IF
	END_IF

15:
	
	PusherServo.xHalt := FALSE;
	tickcounter_Pusher := tickcounter_Pusher + 1;
	IF tickcounter_Pusher >= 10 THEN
		tickcounter_Pusher := 0;
		StateNext := 20;
		//Executed := TRUE;
	END_IF
20:
	PusherServo.fHomeOffset := 0;
	PusherServo.xZero := TRUE;
	StateNext := 25;	
	
25:
	IF PusherServo.xZeroed THEN
		PusherServo.xZero := FALSE;
		_ExecutedHome := TRUE;
		StateNext := 0;
	END_IF
	

END_CASE

State := StateNext;
END_METHOD

METHOD _mc_stop : BOOL
VAR_INPUT
END_VAR
PusherServo.xStop:=TRUE;
END_METHOD

METHOD _Reset
VAR_INPUT
END_VAR
	tickcounter_Pusher:=0;
	PusherServoEnable := FALSE;
	PusherServo.xZero := FALSE;
	PusherServo.xMoveV := FALSE;
	PusherServo.xMoveA := FALSE;
	PusherServo.xMoveR := FALSE;
	PusherServo.xHalt:=FALSE;
	PusherServo.xStop:=FALSE;
	PusherServo.GearIn := FALSE;
	state:=0;
	statenext:=0;
	tickcounter_pusher     :=0;
	
	Stage2Executed:=FALSE;
	Stage4Executed:=FALSE;
	Stage5Executed:=FALSE;
	_ExecutedHome:=FALSE;
	_ExecutedOffset:=FALSE;
END_METHOD

METHOD _Reset_medium
VAR_INPUT
END_VAR
	tickcounter_Pusher:=0;
	PusherServoEnable := FALSE;
	PusherServo.xZero := FALSE;
	PusherServo.xMoveV := FALSE;
	PusherServo.xMoveA := FALSE;
	PusherServo.xMoveR := FALSE;
	PusherServo.xHalt:=FALSE;
	PusherServo.xStop:=FALSE;
	PusherServo.GearIn := FALSE;
	state:=0;
	statenext:=0;
	tickcounter_pusher     :=0;
	
	Stage2Executed:=FALSE;
	Stage4Executed:=FALSE;
	Stage5Executed:=FALSE;
	//_ExecutedHome:=FALSE;
	//_ExecutedOffset:=FALSE;
END_METHOD

METHOD _Soft_Reset
VAR_INPUT
END_VAR

tickcounter_Pusher:=0;
PusherServo.xZero := FALSE;
PusherServo.xMoveV := FALSE;
PusherServo.xMoveA := FALSE;
PusherServo.xHalt := FALSE;
PusherServo.GearIn := FALSE;
PusherServo.xStop:=FALSE;
state:=0;
END_METHOD

METHOD _Stage2 : BOOL
VAR_INPUT
END_VAR
CASE State OF
	
0:	
	_ExecutedStage2:=FALSE;
	PusherServo.fPosition:= _Pusher_Param.Pusher.Initial_Distance;
	PusherServo.fVelocity:= _Pusher_Param.Pusher.Initial_Speed; //mm/s
	PusherServo.xMoveA:=TRUE;
	StateNext:=5;
5:	
	IF PusherServo.xInPosition = TRUE THEN
		
		PusherServo.xMoveA := FALSE;
		StateNext:=0;
		_ExecutedStage2:=TRUE;
		
	END_IF


END_CASE

State:=StateNext;
END_METHOD

METHOD _Stage4
VAR_INPUT
END_VAR

VAR
	
END_VAR
CASE State OF
	
0:	
	
	
	_ExecutedStage4:=FALSE;
	PusherServo.fPosition:= _Pusher_Param.Pusher.Eject_Distance;
	PusherServo.fVelocity:= _Pusher_Param.Pusher.Eject_Speed; //mm/s
	
	_Pusher_Param.Clamp.Release_Instance := _Pusher_Param.Clamp.Release_Instance - _Pusher_Param.Pusher.tamp_final_distance;
		
	IF _Pusher_Param.Clamp.Release_Instance <= 0 THEN
		IF qxClamp = TRUE THEN
			qxClamp:=FALSE;
		
			
			PRG_Machine.StopClampTimer();
	
		END_IF
	END_IF
	
	pusher_old_position:= PusherServo.fActualPosition;
	PusherServo.xMoveA:=TRUE;
	StateNext:=5;
	
5:	
	IF PusherServo.xInPosition = TRUE THEN
		
		PusherServo.xMoveA := FALSE;
		StateNext:=0;
		_ExecutedStage4:=TRUE;
		
		IF qxClamp = TRUE THEN
			qxClamp:=FALSE;
		
			PRG_Machine.StopClampTimer();
	
		END_IF
		
	END_IF
	
	IF (PusherServo.fActualPosition-pusher_old_position) >= (_Pusher_Param.Clamp.Release_Instance) THEN
		IF qxClamp = TRUE THEN
			qxClamp:=FALSE;
		
			PRG_Machine.StopClampTimer();
	
		END_IF
	END_IF


END_CASE

State:=StateNext;
END_METHOD

METHOD _Stage5
VAR_INPUT
END_VAR
CASE State OF
	
0:	
	_ExecutedStage5:=FALSE;
	PusherServo.fPosition:= 0;
	PusherServo.fVelocity:= _Pusher_Param.Pusher.Retract_Speed; //mm/s
	
	PusherServo.xMoveA:=TRUE;
	StateNext:=5;
5:	
	IF PusherServo.xInPosition = TRUE THEN
		
		PusherServo.xMoveA := FALSE;
		StateNext:=0;
		_ExecutedStage5:=TRUE;
		
	END_IF


END_CASE

State:=StateNext;
END_METHOD

METHOD _Update
VAR_INPUT
END_VAR
PusherServo(
	xEnable:= PusherServoEnable, 
	xZero:= , 
	xMoveR:= , 
	xMoveA:= , 
	xMoveV:= , 
	xPositiveDirection:= , 
	fDistance:= , 
	fPosition:= , 
	fVelocity:= , 
	xStop:= , 
	xHome:= , 
	xHomeFlag:= , 
	homePosition:=0,
	fActualPosition=> , 
	fActualVelocity=> , 
	fActModuloPos=> , 
	xEnabled=> PusherServoEnabled, 
	xMoveComplete=> , 
	xInPosition=> , 
	xAtSpeed=> , 
	xStopped=> , 
	xHomed=> ,
	errorID=> PusherServoErrorID, 
	Axis:= PusherAxis );
END_METHOD

PROPERTY HomeExecuted : BOOL
GET
HomeExecuted := _ExecutedHome;
END_GET
SET
_ExecutedHome := HomeExecuted;
END_SET
END_PROPERTY

METHOD Offset
VAR_INPUT
END_VAR
CASE State OF
	
0:	
	_ExecutedOffset:=FALSE;
	PusherServo.fPosition:= _Pusher_Param.Other.Pusher_Home_Offset;
	PusherServo.fVelocity:= 20; //mm/s
	
	IF PusherServo.fPosition<>0 THEN
		PusherServo.xMoveA:=TRUE;
		StateNext:=5;
	ELSE
		_ExecutedOffset:=TRUE;
	END_IF	
	
	//StateNext:=5;
5:	
	IF PusherServo.xInPosition = TRUE THEN
		
		PusherServo.xMoveA := FALSE;
		StateNext:=10;
		//_ExecutedOffset:=TRUE;
		
	END_IF
	
10:
	
	pusherServo.fHomeOffset := 0;
	pusherServo.xZero := TRUE;
	StateNext := 15;	
	
15:
	IF pusherServo.xZeroed THEN
		pusherServo.xZero := FALSE;
		_ExecutedOffset:=TRUE;
		StateNext := 0;
	END_IF


END_CASE

State:=StateNext;
END_METHOD

PROPERTY OffsetExecuted : BOOL
GET
OffsetExecuted := _ExecutedOffset;
END_GET
SET
_ExecutedOffset := OffsetExecuted;
END_SET
END_PROPERTY

PROPERTY Pusher_Param : recipe
GET
Pusher_param := _Pusher_Param;
END_GET
SET
_Pusher_param := Pusher_Param;
END_SET
END_PROPERTY

PROPERTY Stage2Executed : BOOL
GET
Stage2Executed := _ExecutedStage2;
END_GET
SET
_ExecutedStage2 := Stage2Executed;
END_SET
END_PROPERTY

PROPERTY Stage4Executed : BOOL
GET
Stage4Executed := _ExecutedStage4;
END_GET
SET
_ExecutedStage4 := Stage4Executed;
END_SET
END_PROPERTY

PROPERTY Stage5Executed : BOOL
GET
Stage5Executed := _ExecutedStage5;
END_GET
SET
_ExecutedStage5 := Stage5Executed;
END_SET
END_PROPERTY

METHOD Tamp
VAR_INPUT
END_VAR

CASE State OF
	
0:	
	_ExecutedTamp:=FALSE;
	PusherServo.fPosition:= _Pusher_Param.Pusher.tamp_initial_distance;
	PusherServo.fVelocity:= _Pusher_Param.Pusher.tamp_initial_speed;
	
	
	IF  _Pusher_Param.Pusher.tamp_initial_speed = 0 THEN
		StateNext:=10;
	ELSE
		StateNext:=5;
		PusherServo.xMoveA:=TRUE;
	END_IF
	
5:	
	IF PusherServo.xInPosition = TRUE THEN
		
		PusherServo.xMoveA := FALSE;
		StateNext:=10;
	END_IF

10:
	PusherServo.fVelocity:= _Pusher_Param.Pusher.tamp_final_speed;
	PusherServo.fPosition:= _Pusher_Param.Pusher.tamp_final_distance;
	
	
	IF _Pusher_Param.Pusher.tamp_final_speed = 0 THEN
		StateNext:=0;
		_ExecutedTamp:=TRUE;
		
	ELSE
		StateNext:=15;
		PusherServo.xMoveA := TRUE;
	END_IF
	
	
	
	
15:
	IF PusherServo.xInPosition = TRUE THEN
		
		PusherServo.xMoveA := FALSE;
		StateNext:=0;
		_ExecutedTamp:=TRUE;
	END_IF

	

END_CASE

State:=StateNext;
END_METHOD

PROPERTY TampExecuted : BOOL
GET
TampExecuted := _ExecutedTamp;
END_GET
SET
_ExecutedTamp := TampExecuted;
END_SET
END_PROPERTY

END_FUNCTION_BLOCK

// ---- POUs/FB_AxisControl.TcPOU
FUNCTION_BLOCK FB_AxisControl
VAR_INPUT
	xEnable: BOOL;
	xZero: BOOL;
	xMoveR: BOOL;
	xMoveA: BOOL;
	xMoveV: BOOL;
	xPositiveDirection: BOOL;
	fDistance: LREAL;
	fPosition: LREAL;
	fVelocity: LREAL;
	xStop: BOOL;
	xHome: BOOL;
	xHomeFlag: BOOL;
	xHalt: BOOL;
	xTimerInput: BOOL;
	timerPT: TIME;
	HomePosition: LREAL;
	fAxisAcceleration: LREAL;
	fAxisDeceleration: LREAL;
	fAxisJerk: LREAL;
	MasterAxis: AXIS_REF;
	GearIn: BOOL;
	Gear_out: BOOL;
	GearRatio: LREAL;
	EnableSoE_ReadPosition: BOOL;
	EnableSoE_ReadTorque: BOOL;
	EnableSoE_ReadFollowingError: BOOL;
	fHomeOffset: LREAL;
END_VAR
VAR_OUTPUT
	gear_out_busy	:BOOL;
	fActualPosition: LREAL;
	fActualVelocity: LREAL;
	fActModuloPos: LREAL;
	fActPosition: DINT;
	fActFollowingError: DINT;
	fActualTorque: INT;
	xEnabled: BOOL;
	xMoveComplete: BOOL;
	xInPosition: BOOL;
	xAtSpeed: BOOL;
	xStopped: BOOL;
	xHomed: BOOL;
	xHalted: BOOL;
	errorID: UDINT;
	xAxisHomed: BOOL;
	xZeroed: BOOL;
	timerET: TIME;
	timerQOutput: BOOL;
	InGear: BOOL;
	xServoError: BOOL;
	iErrorID: UDINT;
END_VAR
VAR
	mcPower: MC_Power;
	mcReset: MC_Reset;
	mcMoveRelative: MC_MoveRelative;
	mcSetPosition: MC_SetPosition;
	mcMoveAbsolute: MC_MoveAbsolute;
	mcReadStatus: MC_ReadStatus;
	mcMoveVelocity: MC_MoveVelocity;
	mcStop: MC_Stop;
	mcHome: MC_Home;
	mcHalt: MC_Halt;
	timerOn: TON;

	mcGearInDyn: MC_GearInDyn;
	mcGearOut: MC_GearOut;
	
	EnReadPosition: BOOL;
	EnReadTorque: BOOL;
	EnReadFollowingError: BOOL;
	
END_VAR
VAR_IN_OUT
	Axis: AXIS_REF;
	//MasterAxis : AXIS_REF;
END_VAR

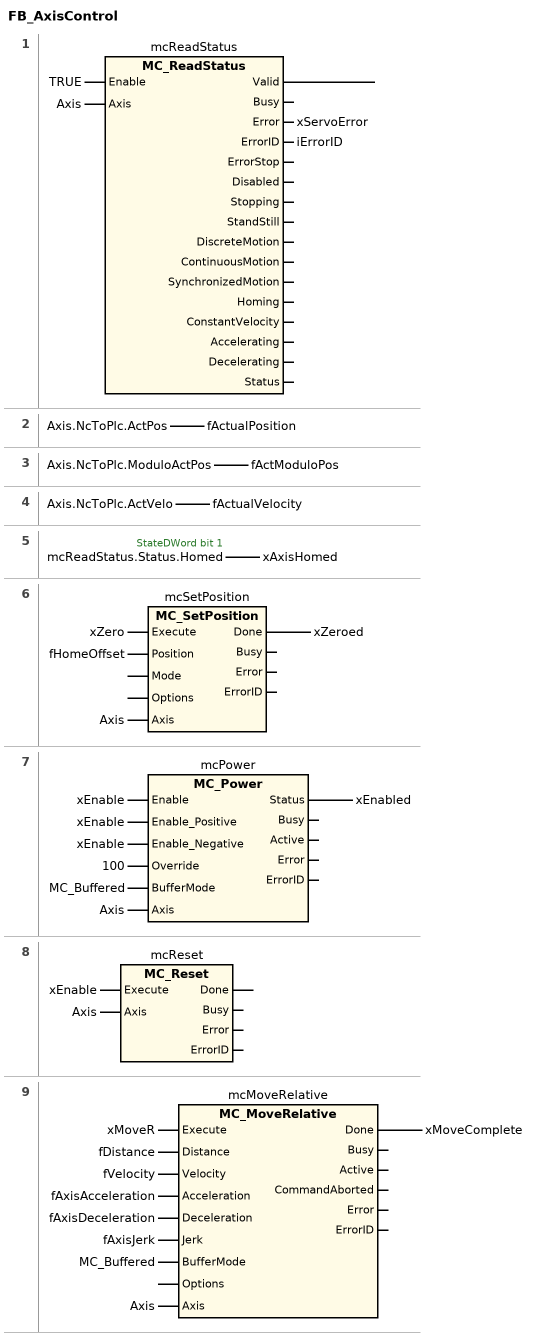
// NETWORK 1
mcReadStatus(Enable := TRUE, Axis := Axis, Error => xServoError, ErrorID => iErrorID); // MC_ReadStatus

// NETWORK 2
fActualPosition := Axis.NcToPlc.ActPos;

// NETWORK 3
fActModuloPos := Axis.NcToPlc.ModuloActPos;

// NETWORK 4
fActualVelocity := Axis.NcToPlc.ActVelo;

// NETWORK 5
//   mcReadStatus.Status.Homed: StateDWord bit 1
xAxisHomed := mcReadStatus.Status.Homed;

// NETWORK 6
mcSetPosition(Execute := xZero, Position := fHomeOffset, Axis := Axis); // MC_SetPosition
xZeroed := mcSetPosition.Done;

// NETWORK 7
mcPower(
    Enable := xEnable,
    Enable_Positive := xEnable,
    Enable_Negative := xEnable,
    Override := 100,
    BufferMode := MC_Buffered,
    Axis := Axis); // MC_Power
xEnabled := mcPower.Status;

// NETWORK 8
mcReset(Execute := xEnable, Axis := Axis); // MC_Reset

// NETWORK 9
mcMoveRelative(
    Execute := xMoveR,
    Distance := fDistance,
    Velocity := fVelocity,
    Acceleration := fAxisAcceleration,
    Deceleration := fAxisDeceleration,
    Jerk := fAxisJerk,
    BufferMode := MC_Buffered,
    Axis := Axis); // MC_MoveRelative
xMoveComplete := mcMoveRelative.Done;

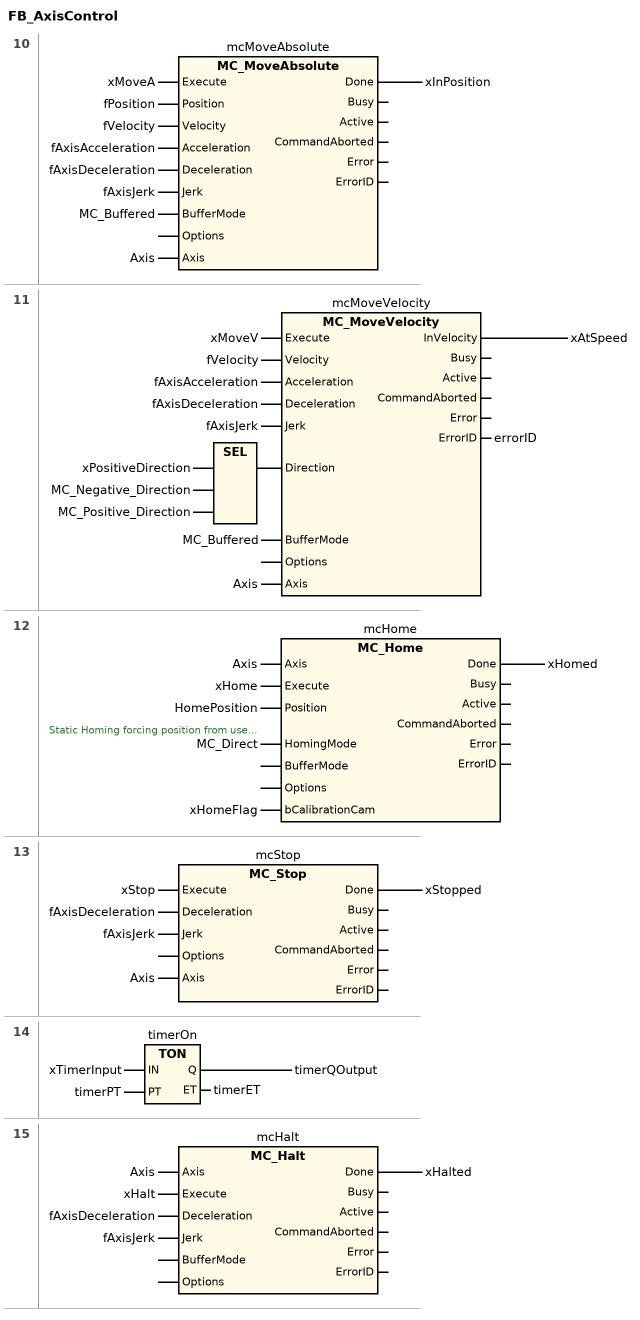
// NETWORK 10
mcMoveAbsolute(
    Execute := xMoveA,
    Position := fPosition,
    Velocity := fVelocity,
    Acceleration := fAxisAcceleration,
    Deceleration := fAxisDeceleration,
    Jerk := fAxisJerk,
    BufferMode := MC_Buffered,
    Axis := Axis); // MC_MoveAbsolute
xInPosition := mcMoveAbsolute.Done;

// NETWORK 11
mcMoveVelocity(
    Execute := xMoveV,
    Velocity := fVelocity,
    Acceleration := fAxisAcceleration,
    Deceleration := fAxisDeceleration,
    Jerk := fAxisJerk,
    Direction := SEL(xPositiveDirection, MC_Negative_Direction, MC_Positive_Direction),
    BufferMode := MC_Buffered,
    Axis := Axis,
    ErrorID => errorID); // MC_MoveVelocity
xAtSpeed := mcMoveVelocity.InVelocity;

// NETWORK 12
//   MC_Direct: Static Homing forcing position from user reference
mcHome(
    Axis := Axis,
    Execute := xHome,
    Position := HomePosition,
    HomingMode := MC_Direct,
    bCalibrationCam := xHomeFlag); // MC_Home
xHomed := mcHome.Done;

// NETWORK 13
mcStop(Execute := xStop, Deceleration := fAxisDeceleration, Jerk := fAxisJerk, Axis := Axis); // MC_Stop
xStopped := mcStop.Done;

// NETWORK 14
timerOn(IN := xTimerInput, PT := timerPT, ET => timerET); // TON
timerQOutput := timerOn.Q;

// NETWORK 15
mcHalt(Axis := Axis, Execute := xHalt, Deceleration := fAxisDeceleration, Jerk := fAxisJerk); // MC_Halt
xHalted := mcHalt.Done;

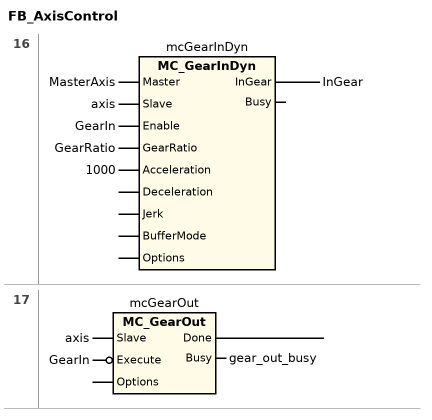
// NETWORK 16
mcGearInDyn(
    Master := MasterAxis,
    Slave := axis,
    Enable := GearIn,
    GearRatio := GearRatio,
    Acceleration := 1000); // MC_GearInDyn
InGear := mcGearInDyn.InGear;

// NETWORK 17
mcGearOut(Slave := axis, Execute := NOT GearIn, Busy => gear_out_busy); // MC_GearOut

END_FUNCTION_BLOCK

// ---- Classes/Compress/FB_Compress.TcPOU
FUNCTION_BLOCK FB_Compress
VAR_INPUT
END_VAR
VAR_OUTPUT
END_VAR
VAR

CompressServo: 				FB_AxisControl;

_Compress_param				:recipe;


ToolPositioningSpeed	: LREAL := 20;
ToolPositioningAccel	: LREAL := 100;
ToolPositioningJerk		: LREAL := 1000;
ToolHomingSpeed			: LREAL := 2;

CompressServoEnable:		BOOL;
CompressServoEnabled:		BOOL;

_ExecutedHome:				BOOL:=FALSE;
_ExecutedStage1:			BOOL:=FALSE;
_ExecutedStage5:			BOOL:=FALSE;
_ExecutedOffset:			BOOL:=FALSE;				

tickcounter_compress: 		INT :=0;
State: 						INT:= 0;
StateNext: 					INT:= 0;
			
	

END_VAR

METHOD _Enable 
VAR_INPUT
END_VAR

CompressServoEnable := TRUE;
END_METHOD

METHOD _Halt : BOOL
VAR_INPUT
END_VAR
CompressServo.xHalt:=TRUE;
END_METHOD

METHOD _Halt_false : BOOL
VAR_INPUT
END_VAR
CompressServo.xHalt:=FALSE;
END_METHOD

METHOD _Home : BOOL
VAR_INPUT
	
END_VAR


VAR

	
	
END_VAR

VAR_OUTPUT
	
END_VAR
CASE State OF //you are here

0:	
	_ExecutedHome := FALSE;
	CompressServo.fVelocity := ToolPositioningSpeed;
	CompressServo.fAxisAcceleration := ToolPositioningAccel;
	CompressServo.fAxisDeceleration := ToolPositioningAccel;
	CompressServo.fAxisJerk := ToolPositioningJerk;

	IF ixCompressHomeSwitch THEN
		CompressServo.xPositiveDirection := FALSE;
		IF  tickcounter_compress < 10 THEN
			tickcounter_compress := tickcounter_compress + 1;  // can be put in onditional
		
		ELSE
		//IF tickcounter_compress >= 10 THEN
			CompressServo.xMoveV := TRUE;
		END_IF
	ELSE
	
		//CompressServo.xHalt := NOT CompressServo.xHalt;
		CompressServo.xMoveV := FALSE;
		//CompressServo.xHalt := NOT CompressServo.xHalt;
		CompressServo.xHalt := TRUE;
		IF CompressServo.xHalted THEN
			tickcounter_compress:=0;
			StateNext := 5;
		END_IF
	
	END_IF
	
5:
	
	CompressServo.xHalt := FALSE;
	tickcounter_compress := tickcounter_compress + 1;
	IF tickcounter_compress >= 10 THEN
		tickcounter_compress := 0;
		StateNext := 10;
	END_IF
	
10:
	CompressServo.fVelocity := ToolHomingSpeed;
	
	IF NOT ixCompressHomeSwitch THEN
		CompressServo.xPositiveDirection := TRUE;
		IF tickcounter_compress < 10 THEN
			tickcounter_compress := tickcounter_compress + 1;
		ELSE
		//IF tickcounter >= 10 THEN
			CompressServo.xMoveV := TRUE;
		END_IF
	ELSE
		CompressServo.xMoveV := FALSE;
		CompressServo.xHalt := TRUE;
		IF CompressServo.xHalted THEN
			tickcounter_compress := 0;
			StateNext := 15;
		END_IF
	END_IF

15:
	
	CompressServo.xHalt := FALSE;
	tickcounter_compress := tickcounter_compress + 1;
	IF tickcounter_compress >= 10 THEN
		tickcounter_compress := 0;
		StateNext := 20;
		//Executed := TRUE;
	END_IF	

20:
	CompressServo.fHomeOffset := 0;
	CompressServo.xZero := TRUE;
	StateNext := 25;	
	
25:
	IF CompressServo.xZeroed THEN
		CompressServo.xZero := FALSE;
		_ExecutedHome := TRUE;
		StateNext := 0;
	END_IF

END_CASE

State := StateNext;
END_METHOD

METHOD _mc_stop : BOOL
VAR_INPUT
END_VAR
CompressServo.xStop:=TRUE;
END_METHOD

METHOD _Reset
VAR_INPUT
END_VAR
	tickcounter_compress:=0;
	CompressServoEnable := FALSE;
	CompressServo.xZero := FALSE;
	CompressServo.xMoveV := FALSE;
	CompressServo.xMoveA := FALSE;
	CompressServo.xHALT:=FALSE;
	CompressServo.xStop:=FALSE;
	CompressServo.GearIn := FALSE;
	state:=0;
	statenext:=0;
	tickcounter_compress     :=0;
	
	Stage1Executed:=FALSE;
	Stage5Executed:=FALSE;
	_ExecutedHome:=FALSE;
	_ExecutedOffset:=FALSE;
END_METHOD

METHOD _Reset_medium
VAR_INPUT
END_VAR
	tickcounter_compress:=0;
	CompressServoEnable := FALSE;
	CompressServo.xZero := FALSE;
	CompressServo.xMoveV := FALSE;
	CompressServo.xMoveA := FALSE;
	CompressServo.xHALT:=FALSE;
	CompressServo.xStop:=FALSE;
	CompressServo.GearIn := FALSE;
	state:=0;
	statenext:=0;
	tickcounter_compress     :=0;
	
	Stage1Executed:=FALSE;
	Stage5Executed:=FALSE;
	//_ExecutedHome:=FALSE;
	//_ExecutedOffset:=FALSE;
END_METHOD

METHOD _Soft_Reset
VAR_INPUT
END_VAR

tickcounter_compress:=0;
CompressServo.xZero := FALSE;
CompressServo.xMoveV := FALSE;
CompressServo.xMoveA := FALSE;
CompressServo.xHalt := FALSE;
CompressServo.GearIn := FALSE;
CompressServo.xStop:=FALSE;
state:=0;
END_METHOD

METHOD _Stage1 
VAR_INPUT
END_VAR
VAR

END_VAR

CASE State OF
	
0:	
	_ExecutedStage1:=FALSE;
	CompressServo.fPosition:= _Compress_Param.Compress.Initial_Distance;
	CompressServo.fVelocity:= _Compress_Param.Compress.Initial_Speed;
	CompressServo.xMoveA:=TRUE;
	StateNext:=5;
5:	
	IF CompressServo.xInPosition = TRUE THEN
		
		CompressServo.xMoveA := FALSE;
		StateNext:=10;
	END_IF

10:
	CompressServo.fVelocity:= _Compress_Param.Compress.Initial_Speed;
	CompressServo.fPosition:= _Compress_Param.Compress.Relax_Distance;
	CompressServo.xMoveA := TRUE;
	StateNext:=15;
	
15:
	IF CompressServo.xInPosition = TRUE THEN
		
		CompressServo.xMoveA := FALSE;
		StateNext:=0;
		_ExecutedStage1:=TRUE;
	END_IF

	

END_CASE

State:=StateNext;
END_METHOD

METHOD _Stage5
VAR_INPUT
END_VAR
CASE State OF
	
0:	
	_ExecutedStage5:=FALSE;
	CompressServo.fPosition:= 0;
	CompressServo.fVelocity:= _Compress_Param.Compress.Retract_Speed; //mm/s
	CompressServo.xMoveA:=TRUE;
	StateNext:=5;
5:	
	IF CompressServo.xInPosition = TRUE THEN
		
		CompressServo.xMoveA := FALSE;
		StateNext:=0;
		_ExecutedStage5:=TRUE;
		
	END_IF


END_CASE

State:=StateNext;
END_METHOD

METHOD _Update
VAR_INPUT
END_VAR
CompressServo(
	xEnable:= CompressServoEnable, 
	xZero:= , 
	xMoveR:= , 
	xMoveA:= , 
	xMoveV:= , 
	xPositiveDirection:= , 
	fDistance:= , 
	fPosition:= , 
	fVelocity:= , 
	xStop:= , 
	xHome:= , 
	xHomeFlag:= , 
	homePosition:=0,
	fActualPosition=> , 
	fActualVelocity=> , 
	fActModuloPos=> , 
	xEnabled=> CompressServoEnabled, 
	xMoveComplete=> , 
	xInPosition=> , 
	xAtSpeed=> , 
	xStopped=> , 
	xHomed=> ,
	errorID=> CompressServoErrorID, 
	Axis:= CompressAxis );
END_METHOD

PROPERTY Compress_Param : recipe
GET
Compress_param := _Compress_Param;
END_GET
SET
_Compress_param := Compress_Param;
END_SET
END_PROPERTY

PROPERTY HomeExecuted : BOOL
GET
HomeExecuted := _ExecutedHome;
END_GET
SET
_ExecutedHome := HomeExecuted;
END_SET
END_PROPERTY

METHOD Offset
VAR_INPUT
END_VAR
CASE State OF
	
0:	
	_ExecutedOffset:=FALSE;
	CompressServo.fPosition:= _Compress_Param.Other.Compress_Home_Offset;
	CompressServo.fVelocity:= 20; //mm/s
	
	IF CompressServo.fPosition<>0 THEN
		CompressServo.xMoveA:=TRUE;
		StateNext:=5;
	ELSE
		_ExecutedOffset:=TRUE;
	END_IF
	
	//StateNext:=5;
5:	
	IF CompressServo.xInPosition = TRUE THEN
		
		CompressServo.xMoveA := FALSE;
		StateNext:=10;
		//_ExecutedOffset:=TRUE;
		
	END_IF
10:
	
	compressServo.fHomeOffset := 0;
	compressServo.xZero := TRUE;
	StateNext := 15;	
	
15:
	IF compressServo.xZeroed THEN
		compressServo.xZero := FALSE;
		_ExecutedOffset:=TRUE;
		StateNext := 0;
	END_IF

END_CASE

State:=StateNext;
END_METHOD

PROPERTY OffsetExecuted : BOOL
GET
OffsetExecuted := _ExecutedOffset;
END_GET
SET
_ExecutedOffset := OffsetExecuted;
END_SET
END_PROPERTY

PROPERTY Stage1Executed : BOOL
GET
Stage1Executed := _ExecutedStage1;
END_GET
SET
_ExecutedStage1 := Stage1Executed;
END_SET
END_PROPERTY

PROPERTY Stage5Executed : BOOL
GET
Stage5Executed := _ExecutedStage5;
END_GET
SET
_ExecutedStage5 := Stage5Executed;
END_SET
END_PROPERTY

END_FUNCTION_BLOCK

// ---- Classes/Shield/FB_Shield.TcPOU
FUNCTION_BLOCK FB_Shield
VAR_INPUT
END_VAR
VAR_OUTPUT
END_VAR
VAR

ShieldServo: 		FB_AxisControl;

_Shield_param				:recipe;

distance1:					LREAL:=67;




ToolPositioningSpeed	: LREAL := 20;
ToolPositioningAccel	: LREAL := 100;
ToolPositioningJerk		: LREAL := 1000;
ToolHomingSpeed			: LREAL := 2;

ShieldServoEnable:  BOOL;
ShieldServoEnabled: BOOL;

_ExecutedHome				:BOOL:=FALSE;
_ExecutedStage2 			:BOOL:=FALSE;
_ExecutedStage3				:BOOL:=FALSE;
_ExecutedOffset				:BOOL:=FALSE;

tickcounter_shield: 		INT :=0;
State: 						INT:= 0;
StateNext: 					INT:= 0;

END_VAR

METHOD _Enable 
VAR_INPUT
END_VAR

ShieldServoEnable := TRUE;
END_METHOD

METHOD _Halt : BOOL
VAR_INPUT
END_VAR
ShieldServo.xHalt:=TRUE;
END_METHOD

METHOD _Halt_false : BOOL
VAR_INPUT
END_VAR
ShieldServo.xHalt:=FALSE;
END_METHOD

METHOD _Home 
VAR_INPUT
	
END_VAR


VAR



END_VAR

VAR_OUTPUT
	
END_VAR





CASE State OF //you are here



0:	
	_ExecutedHome := FALSE;
	ShieldServo.fVelocity := ToolPositioningSpeed;
	ShieldServo.fAxisAcceleration := ToolPositioningAccel;
	ShieldServo.fAxisDeceleration := ToolPositioningAccel;
	ShieldServo.fAxisJerk := ToolPositioningJerk;

	IF ixShieldHomeSwitch THEN
		ShieldServo.xPositiveDirection := FALSE;
		IF  tickcounter_shield < 10 THEN
			tickcounter_shield := tickcounter_shield + 1;  // can be put in onditional
		
		ELSE
		//IF tickcounter_compress >= 10 THEN
			ShieldServo.xMoveV := TRUE;
		END_IF
	ELSE
	
		//CompressServo.xHalt := NOT CompressServo.xHalt;
		ShieldServo.xMoveV := FALSE;
		//CompressServo.xHalt := NOT CompressServo.xHalt;
		ShieldServo.xHalt := TRUE;
		IF ShieldServo.xHalted THEN
			tickcounter_shield:=0;
			StateNext := 5;
		END_IF
	
	END_IF
	
5:
	
	ShieldServo.xHalt := FALSE;
	tickcounter_shield := tickcounter_shield + 1;
	IF tickcounter_shield >= 10 THEN
		tickcounter_shield := 0;
		StateNext := 10;
	END_IF
	
10:
	ShieldServo.fVelocity := ToolHomingSpeed;
	
	IF NOT ixShieldHomeSwitch THEN
		ShieldServo.xPositiveDirection := TRUE;
		IF tickcounter_shield < 10 THEN
			tickcounter_shield := tickcounter_shield + 1;
		ELSE
		//IF tickcounter >= 10 THEN
			shieldServo.xMoveV := TRUE;
		END_IF
	ELSE
		shieldServo.xMoveV := FALSE;
		shieldServo.xHalt := TRUE;
		IF shieldServo.xHalted THEN
			tickcounter_shield := 0;
			StateNext := 15;
		END_IF
	END_IF

15:
	
	shieldServo.xHalt := FALSE;
	tickcounter_shield := tickcounter_shield + 1;
	IF tickcounter_shield >= 10 THEN
		tickcounter_shield := 0;
		StateNext := 20;
		//Executed := TRUE;
	END_IF
20:
	shieldServo.fHomeOffset := 0;
	shieldServo.xZero := TRUE;
	StateNext := 25;	
	
25:
	IF shieldServo.xZeroed THEN
		shieldServo.xZero := FALSE;
		_ExecutedHome := TRUE;
		StateNext := 0;
	END_IF
	

END_CASE

State := StateNext;
END_METHOD

METHOD _mc_stop : BOOL
VAR_INPUT
END_VAR
ShieldServo.xStop:=TRUE;
END_METHOD

METHOD _Reset
VAR_INPUT
END_VAR
	tickcounter_Shield:=0;
	ShieldServoEnable := FALSE;
	ShieldServo.xZero := FALSE;
	ShieldServo.xMoveV := FALSE;
	ShieldServo.xMoveA := FALSE;
	ShieldServo.xHalt := FALSE;
	ShieldServo.GearIn := FALSE;
	ShieldServo.xStop:=FALSE;
	state:=0;
	statenext:=0;
	tickcounter_shield     :=0;
	
	Stage2Executed:=FALSE;
	Stage3Executed:=FALSE;
	_ExecutedHome:=FALSE;
	_ExecutedOffset:=FALSE;
END_METHOD

METHOD _Reset_medium
VAR_INPUT
END_VAR
	tickcounter_Shield:=0;
	ShieldServoEnable := FALSE;
	ShieldServo.xZero := FALSE;
	ShieldServo.xMoveV := FALSE;
	ShieldServo.xMoveA := FALSE;
	ShieldServo.xHalt := FALSE;
	ShieldServo.GearIn := FALSE;
	ShieldServo.xStop:=FALSE;
	state:=0;
	statenext:=0;
	tickcounter_shield     :=0;
	
	Stage2Executed:=FALSE;
	Stage3Executed:=FALSE;
END_METHOD

METHOD _Soft_Reset
VAR_INPUT
END_VAR

tickcounter_Shield:=0;
ShieldServo.xZero := FALSE;
ShieldServo.xMoveV := FALSE;
ShieldServo.xMoveA := FALSE;
ShieldServo.xHalt := FALSE;
ShieldServo.GearIn := FALSE;
ShieldServo.xStop:=FALSE;
state:=0;
END_METHOD

METHOD _Stage2 : BOOL
VAR_INPUT
END_VAR
CASE State OF
	
0:	
	_ExecutedStage2:=FALSE;
	ShieldServo.fPosition:= _Shield_Param.Shield.Initial_Distance;
	ShieldServo.fVelocity:= _Shield_Param.Shield.Initial_Speed; //mm/s
	
	
	ShieldServo.xMoveA:=TRUE;
	
	
	StateNext:=5;
5:	
	IF ShieldServo.xInPosition = TRUE THEN
		
		ShieldServo.xMoveA := FALSE;
		StateNext:=0;
		_ExecutedStage2:=TRUE;
		
		
	END_IF


END_CASE

State:=StateNext;
END_METHOD

METHOD _Stage3
VAR_INPUT
END_VAR
CASE State OF
	
0:	
	_ExecutedStage3:=FALSE;
	ShieldServo.fPosition:= 0;
	ShieldServo.fVelocity:= _Shield_Param.Shield.Retract_Speed; //mm/s
	
	
	ShieldServo.xMoveA:=TRUE;
	
	
	StateNext:=5;
5:	
	IF ShieldServo.xInPosition = TRUE THEN
		
		ShieldServo.xMoveA := FALSE;
		StateNext:=0;
		_ExecutedStage3:=TRUE;
		
	END_IF


END_CASE

State:=StateNext;
END_METHOD

METHOD _Update
VAR_INPUT
END_VAR
ShieldServo(
	xEnable:= ShieldServoEnable, 
	xZero:= , 
	xMoveR:= , 
	xMoveA:= , 
	xMoveV:= , 
	xPositiveDirection:= , 
	fDistance:= , 
	fPosition:= , 
	fVelocity:= , 
	xStop:= , 
	xHome:= , 
	xHomeFlag:= , 
	homePosition:=0,
	fActualPosition=> , 
	fActualVelocity=> , 
	fActModuloPos=> , 
	xEnabled=> ShieldServoEnabled, 
	xMoveComplete=> , 
	xInPosition=> , 
	xAtSpeed=> , 
	xStopped=> , 
	xHomed=> ,
	errorID=> ShieldServoErrorID, 
	Axis:= ShieldAxis );
END_METHOD

PROPERTY HomeExecuted : BOOL;
GET
HomeExecuted := _ExecutedHome;
END_GET
SET
_ExecutedHome := HomeExecuted;
END_SET
END_PROPERTY

METHOD Offset
VAR_INPUT
END_VAR
CASE State OF
	
0:	
	_ExecutedOffset:=FALSE;
	ShieldServo.fPosition:= _Shield_Param.Other.Shield_Home_Offset;
	ShieldServo.fVelocity:= 20; //mm/s
	
	IF ShieldServo.fPosition<>0 THEN
		ShieldServo.xMoveA:=TRUE;
		StateNext:=5;
	ELSE
		_ExecutedOffset:=TRUE;
	END_IF
	
	//StateNext:=5;
5:	
	IF ShieldServo.xInPosition = TRUE THEN
		
		ShieldServo.xMoveA := FALSE;
		StateNext:=10;
		//_ExecutedOffset:=TRUE;
		
	END_IF
	
10:
	
	shieldServo.fHomeOffset := 0;
	shieldServo.xZero := TRUE;
	StateNext := 15;	
	
15:
	IF shieldServo.xZeroed THEN
		shieldServo.xZero := FALSE;
		_ExecutedOffset := TRUE;
		StateNext := 0;
	END_IF


END_CASE

State:=StateNext;
END_METHOD

PROPERTY OffsetExecuted : BOOL
GET
OffsetExecuted := _ExecutedOffset;
END_GET
SET
_ExecutedOffset := OffsetExecuted;
END_SET
END_PROPERTY

PROPERTY Shield_Param : recipe
GET
Shield_param := _Shield_Param;
END_GET
SET
_Shield_param := Shield_Param;
END_SET
END_PROPERTY

PROPERTY Stage2Executed : BOOL
GET
Stage2Executed := _ExecutedStage2;
END_GET
SET
_ExecutedStage2 := Stage2Executed;
END_SET
END_PROPERTY

PROPERTY Stage3Executed : BOOL
GET
Stage3Executed := _ExecutedStage3;
END_GET
SET
_ExecutedStage3 := Stage3Executed;
END_SET
END_PROPERTY

END_FUNCTION_BLOCK

// ---- POUs/Config_Slow.TcPOU
PROGRAM Config_Slow
VAR
	
	
	Once				:BOOL :=TRUE;
	saving_config		:BOOL :=FALSE;		
END_VAR

IF Clock.DateTimeInitialised THEN
   	//Config_Counter:=Config_Counter+1;
	//config_count:=config_count+1;
	//IF config_count = 30 THEN
	//	Config();
	//	config_count:=0;
	//END_IF
	IF Config.Initialised() = FALSE THEN
		Config();
	ELSIF Once = TRUE THEN
		Message := 'Data Loaded';
		Once := FALSE;
	END_IF
	
	
	IF Config_Request = TRUE AND saving_config = FALSE THEN
		Config_Request:=FALSE;
		saving_config:=TRUE;
		config_count:=0;

	END_IF
	
	IF saving_config AND config_count <=2500 THEN
		Config();
		config_count:=config_count+1;
	END_IF
	
	IF config_count = 2500 THEN
		saving_config:= FALSE;
		config_count :=0;
		IF config_request = FALSE THEN
			Message := 'Operation Configured';
		END_IF
	END_IF	

END_IF

END_PROGRAM

// ---- POUs/FB_LampController.TcPOU
FUNCTION_BLOCK FB_LampController
VAR_INPUT
	State:E_LampState;
END_VAR
VAR_OUTPUT
	Q : BOOL := FALSE;
END_VAR
VAR
	FlashOffTime: TON;
	FlashOnTime: TON;
	LampFlash: BOOL := TRUE;
END_VAR

FlashOffTime();
FlashOnTime();

//IF NOT Steady AND NOT Flash_Fast AND NOT Flash_Slow THEN 
IF State = 0 THEN
	q := FALSE;
END_IF

//IF Steady AND NOT Flash_Fast AND NOT Flash_Slow THEN 
IF State = 1 THEN
	q := TRUE;
END_IF

//IF NOT Steady AND Flash_Fast AND NOT Flash_Slow THEN 
IF State = 2 THEN
	FlashOffTime.PT := T#250MS;
	FlashOnTime.PT := T#100MS;
END_IF

//IF NOT Steady AND NOT Flash_Fast AND Flash_Slow THEN 
IF State = 4 THEN
	FlashOffTime.PT := T#1500MS;
	FlashOnTime.PT := T#250MS;
END_IF

IF state > 1 THEN 
	IF LampFlash THEN
	 	FlashOnTime.IN := TRUE;
		FlashOffTime.IN := FALSE;
		q := TRUE;
		IF FlashOnTime.Q THEN 
			LampFlash := FALSE;
		END_IF
	ELSE 
		FlashOnTime.IN := FALSE;
		FlashOffTime.IN := TRUE;
		q := FALSE;
		IF FlashOffTime.Q THEN 
			LampFlash := TRUE;
		END_IF
	END_IF
END_IF

IF LampTest THEN
	q := TRUE;
END_IF

END_FUNCTION_BLOCK

// ---- Classes/Config/TConfig.TcPOU
FUNCTION_BLOCK TConfig
VAR
    Recipe_mem_1 						AT %MD0: STRING(20);
	Recipe_mem_2 						AT %MD5: STRING(20);
	Recipe_mem_3 						AT %MD10: STRING(20);
	Recipe_mem_4 						AT %MD15: STRING(20);
	Recipe_mem_5 						AT %MD20: STRING(20);
	Recipe_mem_6 						AT %MD25: STRING(20);
	Recipe_mem_7 						AT %MD30: STRING(20);
	Recipe_mem_8 						AT %MD35: STRING(20);
	Recipe_mem_9 						AT %MD40: STRING(20);
	Recipe_mem_10 						AT %MD45: STRING(20);
	
	Rec1_Name_1								AT %MD0 :UDINT;
	Rec1_Name_2								AT %MD1 :UDINT;
	Rec1_Name_3								AT %MD2 :UDINT;
	Rec1_Name_4								AT %MD3 :UDINT;
	Rec1_Name_5								AT %MD4 :UDINT;
	
	Rec2_Name_1								AT %MD5 :UDINT;
	Rec2_Name_2								AT %MD6 :UDINT;
	Rec2_Name_3								AT %MD7 :UDINT;
	Rec2_Name_4								AT %MD8 :UDINT;
	Rec2_Name_5								AT %MD9 :UDINT;
	
	Rec3_Name_1								AT %MD10 :UDINT;
	Rec3_Name_2								AT %MD11 :UDINT;
	Rec3_Name_3								AT %MD12 :UDINT;
	Rec3_Name_4								AT %MD13 :UDINT;
	Rec3_Name_5								AT %MD14:UDINT;
	
	Rec4_Name_1								AT %MD15 :UDINT;
	Rec4_Name_2								AT %MD16 :UDINT;
	Rec4_Name_3								AT %MD17 :UDINT;
	Rec4_Name_4								AT %MD18 :UDINT;
	Rec4_Name_5								AT %MD19 :UDINT;
	
	Rec5_Name_1								AT %MD20 :UDINT;
	Rec5_Name_2								AT %MD21 :UDINT;
	Rec5_Name_3								AT %MD22 :UDINT;
	Rec5_Name_4								AT %MD23 :UDINT;
	Rec5_Name_5								AT %MD24 :UDINT;
	
	Rec6_Name_1								AT %MD25 :UDINT;
	Rec6_Name_2								AT %MD26 :UDINT;
	Rec6_Name_3								AT %MD27 :UDINT;
	Rec6_Name_4								AT %MD28 :UDINT;
	Rec6_Name_5								AT %MD29 :UDINT;
	
	Rec7_Name_1								AT %MD30 :UDINT;
	Rec7_Name_2								AT %MD31 :UDINT;
	Rec7_Name_3								AT %MD32 :UDINT;
	Rec7_Name_4								AT %MD33 :UDINT;
	Rec7_Name_5								AT %MD34 :UDINT;
	
	Rec8_Name_1								AT %MD35 :UDINT;
	Rec8_Name_2								AT %MD36 :UDINT;
	Rec8_Name_3								AT %MD37 :UDINT;
	Rec8_Name_4								AT %MD38 :UDINT;
	Rec8_Name_5								AT %MD39 :UDINT;
	
	Rec9_Name_1								AT %MD40 :UDINT;
	Rec9_Name_2								AT %MD41 :UDINT;
	Rec9_Name_3								AT %MD42 :UDINT;
	Rec9_Name_4								AT %MD43 :UDINT;
	Rec9_Name_5								AT %MD44 :UDINT;
	
	Rec10_Name_1							AT %MD45 :UDINT;
	Rec10_Name_2							AT %MD46 :UDINT;
	Rec10_Name_3							AT %MD47 :UDINT;
	Rec10_Name_4							AT %MD48 :UDINT;
	Rec10_Name_5							AT %MD49 :UDINT;
	
	PersistentData : TPersistentData;
	
    ConfigData : TConfigData := (
		Other1_Memory_Free := 1,
		Other2_Memory_Free := 1,		
		Other3_Memory_Free := 1,				
		Other4_Memory_Free := 1,
		Other5_Memory_Free := 1,
		Other6_Memory_Free := 1,
		Other7_Memory_Free := 1,
		Other8_Memory_Free := 1,
		Other9_Memory_Free := 1,
		Other10_Memory_Free := 1);		
END_VAR

PersistentData(
	DataAddress:= ADR(ConfigData), 
	DataLength:= SIZEOF(ConfigData), 
	Filename:= 'Hard Disk\TwinCAT\3.1\Boot\Config.txt', 
	Timestamp:= Clock.DateTimeAsString, 
	LoadFromFile:= NOT ConfigData.Initialised, 
	AutoSave:= TRUE, 
	ValuesReadFromFile=> ConfigData.Initialised, 
	Error=> , 
	ErrorId=> , 
	ErrorText=> );

METHOD CopyConfigRecipiesToGlobal : BOOL
VAR_INPUT
END_VAR
//GVL_Objects.List_of_Recipes[1].Name := ConfigData.Rec1_Name;

Rec1_Name_1:=ConfigData.Rec1_Name_1;								
Rec1_Name_2:=ConfigData.Rec1_Name_2;								
Rec1_Name_3:=ConfigData.Rec1_Name_3;								
Rec1_Name_4:=ConfigData.Rec1_Name_4;								
Rec1_Name_5:=ConfigData.Rec1_Name_5;
List_of_Recipes[1].Name := Recipe_mem_1;

GVL_Objects.List_of_Recipes[1].Shield.Retract_Speed := ConfigData.Rec1_Shield_Retract_Speed;
GVL_Objects.List_of_Recipes[1].Shield.Initial_Speed := ConfigData.Rec1_Shield_Initial_Speed;
GVL_Objects.List_of_Recipes[1].Shield.Initial_Distance := ConfigData.Rec1_Shield_Initial_Distance;

GVL_Objects.List_of_Recipes[1].Compress.Initial_Speed :=  ConfigData.Rec1_Compress_Initial_Speed;
GVL_Objects.List_of_Recipes[1].Compress.Initial_Distance := ConfigData.Rec1_Compress_Initial_Distance;
GVL_Objects.List_of_Recipes[1].Compress.Shield_Dwell := ConfigData.Rec1_Compress_Shield_Dwell;
GVL_Objects.List_of_Recipes[1].Compress.Relax_Distance := ConfigData.Rec1_Compress_Relax_Distance;
GVL_Objects.List_of_Recipes[1].Compress.Retract_Speed := ConfigData.Rec1_Compress_Retract_Speed;

GVL_Objects.List_of_Recipes[1].Pusher.Initial_Speed := ConfigData.Rec1_Pusher_Initial_Speed;
GVL_Objects.List_of_Recipes[1].Pusher.Initial_Distance := ConfigData.Rec1_Pusher_Initial_Distance;
GVL_Objects.List_of_Recipes[1].Pusher.Eject_Speed := ConfigData.Rec1_Pusher_Eject_Speed;
GVL_Objects.List_of_Recipes[1].Pusher.Eject_Distance := ConfigData.Rec1_Pusher_Eject_Distance;
GVL_Objects.List_of_Recipes[1].Pusher.Retract_Speed := ConfigData.Rec1_Pusher_Retract_Speed;

GVL_Objects.List_of_Recipes[1].Pusher.tamp_final_distance := ConfigData.Rec1_Pusher_tamp_final_distance;
GVL_Objects.List_of_Recipes[1].Pusher.tamp_final_speed := ConfigData.Rec1_Pusher_tamp_final_speed;
GVL_Objects.List_of_Recipes[1].Pusher.tamp_initial_distance := ConfigData.Rec1_Pusher_tamp_initial_distance;
GVL_Objects.List_of_Recipes[1].Pusher.tamp_initial_speed := ConfigData.Rec1_Pusher_tamp_initial_speed;

GVL_Objects.List_of_Recipes[1].Other.Compress_Home_Offset := ConfigData.Other1_Compress_Home_Offset;
GVL_Objects.List_of_Recipes[1].Other.Pusher_Home_Offset := ConfigData.Other1_Pusher_Home_Offset;
GVL_Objects.List_of_Recipes[1].Other.Shield_Home_Offset := ConfigData.Other1_Shield_Home_Offset;
GVL_Objects.List_of_Recipes[1].Other.Axis_Acceleration := ConfigData.Other1_Axis_Acceleration;
GVL_Objects.List_of_Recipes[1].Other.Axis_Deceleration := ConfigData.Other1_Axis_Deceleration;
GVL_Objects.List_of_Recipes[1].Other.Axis_Jerk := ConfigData.Other1_Axis_Jerk;
GVL_Objects.List_of_Recipes[1].Memory_Free := LREAL_TO_BOOL(ConfigData.Other1_Memory_Free);

GVL_Objects.List_of_Recipes[1].Clamp.Release_Instance := ConfigData.Clamp1_Release_Instance;

//u are here
Rec2_Name_1:=ConfigData.Rec2_Name_1;								
Rec2_Name_2:=ConfigData.Rec2_Name_2;								
Rec2_Name_3:=ConfigData.Rec2_Name_3;								
Rec2_Name_4:=ConfigData.Rec2_Name_4;								
Rec2_Name_5:=ConfigData.Rec2_Name_5;
List_of_Recipes[2].Name := Recipe_mem_2;

GVL_Objects.List_of_Recipes[2].Shield.Retract_Speed := ConfigData.Rec2_Shield_Retract_Speed;
GVL_Objects.List_of_Recipes[2].Shield.Initial_Speed := ConfigData.Rec2_Shield_Initial_Speed;
GVL_Objects.List_of_Recipes[2].Shield.Initial_Distance := ConfigData.Rec2_Shield_Initial_Distance;

GVL_Objects.List_of_Recipes[2].Compress.Initial_Speed :=  ConfigData.Rec2_Compress_Initial_Speed;
GVL_Objects.List_of_Recipes[2].Compress.Initial_Distance := ConfigData.Rec2_Compress_Initial_Distance;
GVL_Objects.List_of_Recipes[2].Compress.Shield_Dwell := ConfigData.Rec2_Compress_Shield_Dwell;
GVL_Objects.List_of_Recipes[2].Compress.Relax_Distance := ConfigData.Rec2_Compress_Relax_Distance;
GVL_Objects.List_of_Recipes[2].Compress.Retract_Speed := ConfigData.Rec2_Compress_Retract_Speed;

GVL_Objects.List_of_Recipes[2].Pusher.Initial_Speed := ConfigData.Rec2_Pusher_Initial_Speed;
GVL_Objects.List_of_Recipes[2].Pusher.Initial_Distance := ConfigData.Rec2_Pusher_Initial_Distance;
GVL_Objects.List_of_Recipes[2].Pusher.Eject_Speed := ConfigData.Rec2_Pusher_Eject_Speed;
GVL_Objects.List_of_Recipes[2].Pusher.Eject_Distance := ConfigData.Rec2_Pusher_Eject_Distance;
GVL_Objects.List_of_Recipes[2].Pusher.Retract_Speed := ConfigData.Rec2_Pusher_Retract_Speed;

GVL_Objects.List_of_Recipes[2].Pusher.tamp_final_distance := ConfigData.Rec2_Pusher_tamp_final_distance;
GVL_Objects.List_of_Recipes[2].Pusher.tamp_final_speed := ConfigData.Rec2_Pusher_tamp_final_speed;
GVL_Objects.List_of_Recipes[2].Pusher.tamp_initial_distance := ConfigData.Rec2_Pusher_tamp_initial_distance;
GVL_Objects.List_of_Recipes[2].Pusher.tamp_initial_speed := ConfigData.Rec2_Pusher_tamp_initial_speed;

GVL_Objects.List_of_Recipes[2].Other.Compress_Home_Offset := ConfigData.Other2_Compress_Home_Offset;
GVL_Objects.List_of_Recipes[2].Other.Pusher_Home_Offset := ConfigData.Other2_Pusher_Home_Offset;
GVL_Objects.List_of_Recipes[2].Other.Shield_Home_Offset := ConfigData.Other2_Shield_Home_Offset;
GVL_Objects.List_of_Recipes[2].Other.Axis_Acceleration := ConfigData.Other2_Axis_Acceleration;
GVL_Objects.List_of_Recipes[2].Other.Axis_Deceleration := ConfigData.Other2_Axis_Deceleration;
GVL_Objects.List_of_Recipes[2].Other.Axis_Jerk := ConfigData.Other2_Axis_Jerk;
GVL_Objects.List_of_Recipes[2].Memory_Free := LREAL_TO_BOOL(ConfigData.Other2_Memory_Free);

GVL_Objects.List_of_Recipes[2].Clamp.Release_Instance := ConfigData.Clamp2_Release_Instance;

Rec3_Name_1:=ConfigData.Rec3_Name_1;								
Rec3_Name_2:=ConfigData.Rec3_Name_2;								
Rec3_Name_3:=ConfigData.Rec3_Name_3;								
Rec3_Name_4:=ConfigData.Rec3_Name_4;								
Rec3_Name_5:=ConfigData.Rec3_Name_5;
List_of_Recipes[3].Name := Recipe_mem_3;

GVL_Objects.List_of_Recipes[3].Shield.Retract_Speed := ConfigData.Rec3_Shield_Retract_Speed;
GVL_Objects.List_of_Recipes[3].Shield.Initial_Speed := ConfigData.Rec3_Shield_Initial_Speed;
GVL_Objects.List_of_Recipes[3].Shield.Initial_Distance := ConfigData.Rec3_Shield_Initial_Distance;

